ACTION Initialize:
// set interface array instances
aTestItems[ii] := ADR(fbTestFileLog);		ii := ii + 1;
aTestItems[ii] := ADR(fbTestSystemInfo); 	ii := ii + 1;
aTestItems[ii] := ADR(fbTestStation); 		ii := ii + 1;

//aTestItems[ii] := ADR(fbTestpid..);	ii := ii + 1;

bInitDone := TRUE;
END_ACTION

END_PROGRAM

// ---- Background/UnitTest/TestCases/Base/FB_TestCaseBase.TcPOU
/// Test case template
FUNCTION_BLOCK INTERNAL FB_TestCaseBase IMPLEMENTS ITestCase
VAR
	/// state of test case
	eState	: E_TestCaseState;
	/// result of test case
	eResult	: E_TestResult;
END_VAR

{attribute 'object_name' := 'Reset'}
METHOD Reset
// reset var's
eState := E_TestCaseState.eTestCaseState_ready;
eResult := E_TestResult.eTestResult_none;
END_METHOD

{attribute 'object_name' := 'Run'}
METHOD Run : E_TestCaseState
// set state to running, if ready
IF eState = E_TestCaseState.eTestCaseState_ready AND eResult = E_TestResult.eTestResult_none THEN
	eState := E_TestCaseState.eTestCaseState_running;
ELSIF eState <> E_TestCaseState.eTestCaseState_running THEN
	eState := E_TestCaseState.eTestCaseState_error;
END_IF

Run := eState;
END_METHOD

{attribute 'monitoring' := 'call'}
PROPERTY TestResult : E_TestResult
GET
TestResult := eResult;
END_GET
END_PROPERTY

{attribute 'monitoring' := 'call'}
PROPERTY TestState : E_TestCaseState
GET
TestState := eState;
END_GET
END_PROPERTY

END_FUNCTION_BLOCK

// ---- Background/UnitTest/TestCases/FB_TestCase01FileLog.TcPOU
FUNCTION_BLOCK FB_TestCase01FileLog EXTENDS FB_TestCaseBase
VAR
	/// dependencies
	ILog: I_Logger;
	
	bTestOk : BOOL := FALSE;
	bAddInfo, bAddWarn, bAddErr : BOOL;
END_VAR

{attribute 'object_name' := 'Run'}
METHOD Run : E_TestCaseState
// init state in base
Run := SUPER^.Run();
IF Run <> E_TestCaseState.eTestCaseState_running THEN
	RETURN;
END_IF

// test
ILog := Services.ILog;

IF bAddInfo THEN
	bAddInfo := FALSE;
	ILog.AddLog('Test none log message', sSource, E_LogLevel.eLogLevel_none);
	ILog.AddLog('Test info log message', sSource, E_LogLevel.eLogLevel_info);
	//P_HMI_Controller.UpdateNotificationPrio(E_Notification.eNotification_generalInf, TRUE, "UnitTest: eNotification_generalInf", E_Priority.ePriority_info);

	//SUPER^.M_SetErrorEx1(stTextListGlobal.stText_NG_Station005,  // Grp
	//				stTextListGlobal.stText_ST005_Name, "Antrieb (+E2-XXU1)", TO_WSTRING(fbDrive[E_St005_Object_Drive.eSt005_Drive_Antrieb].sErrText), 
	//				E_NotificationMode.eNotificationMode_Auto);

END_IF

IF bAddWarn THEN
	bAddWarn := FALSE;
	ILog.AddLog('Test warning log message', sSource, E_LogLevel.eLogLevel_warn);
	//P_HMI_Controller.UpdateNotificationPrio(E_Notification.eNotification_generalWarn, TRUE, "UnitTest: eNotification_generalWarn", E_Priority.ePriority_warning);
END_IF

IF bAddErr THEN
	bAddErr := FALSE;
	ILog.AddLog('Test error log message', sSource, E_LogLevel.eLogLevel_err);
	//P_HMI_Controller.UpdateNotificationPrio(E_Notification.eNotification_generalErr, TRUE, "UnitTest: eNotification_generalErr", E_Priority.ePriority_fault);
END_IF

// update result and state
IF bTestOk	THEN
	bTestOk := FALSE;
	eResult := E_TestResult.eTestResult_ok; //check log files!
	eState := E_TestCaseState.eTestCaseState_finished;
	Run := eState;
END_IF
END_METHOD

END_FUNCTION_BLOCK

// ---- Background/UnitTest/TestCases/FB_TestCase02SystemInfo.TcPOU
FUNCTION_BLOCK FB_TestCase02SystemInfo EXTENDS FB_TestCaseBase
VAR
	stTestPlcSystemInfo: ST_PlcSystemInfo;
	bTestOk : BOOL := TRUE;
END_VAR

{attribute 'object_name' := 'Run'}
METHOD Run : E_TestCaseState
// init state in base
Run := SUPER^.Run();
IF Run <> E_TestCaseState.eTestCaseState_running THEN
	RETURN;
END_IF

// test
stTestPlcSystemInfo := Statics.stPlcSystemInfo;

// update result and state
IF bTestOk THEN
	eResult := E_TestResult.eTestResult_ok; //check stTestPlcSystemInfo
	eState := E_TestCaseState.eTestCaseState_finished;
END_IF

Run := eState;
END_METHOD

END_FUNCTION_BLOCK

// ---- Background/UnitTest/TestCases/FB_TestCase03Station.TcPOU
FUNCTION_BLOCK FB_TestCase03Station EXTENDS FB_TestCaseBase
VAR
	fbTestStation	: FB_TestStation;
	stTestStationIO : ST_TestStation_IO;
	eStState		: E_ComponentState;
	iTest			: INT;
	bInit			: BOOL;
	bEnable			: BOOL := TRUE;
	bSafetyOk		: BOOL := TRUE;
	bTestOk 		: BOOL := FALSE;
END_VAR

{attribute 'object_name' := 'Run'}
METHOD Run : E_TestCaseState
// init state in base
Run := SUPER^.Run();
IF Run <> E_TestCaseState.eTestCaseState_running THEN
	RETURN;
END_IF

// test
fbTestStation.Enable := bEnable;
fbTestStation.SafetyOk := bSafetyOk;
fbTestStation();
CASE iTest OF
	0:	// init / idle / no Test
		IF NOT bInit THEN
			iTest := 1;
			RETURN;
		END_IF
		
	10:	// init Station
		bInit := TRUE;
		fbTestStation.stIO := stTestStationIO;		
		
	20:	// reset
		fbTestStation.Reset();
		
	30:	// execute command
		;//stRes := fbTestStation.ExecuteCmd(stCmd);
		
END_CASE
iTest := 0;

// update result and state
IF bTestOk THEN
	eResult := E_TestResult.eTestResult_ok; //check log files!
	eState := E_TestCaseState.eTestCaseState_finished;
END_IF

Run := eState;
END_METHOD

END_FUNCTION_BLOCK

// ---- Background/UnitTest/TestCases/StationTest/FB_TestStation.TcPOU
FUNCTION_BLOCK FB_TestStation EXTENDS FB_StationBase
VAR_INPUT
	// IO ref
	stIO	: REFERENCE TO ST_TestStation_IO;
END_VAR
VAR_OUTPUT
END_VAR
VAR
	// components
	fbAxis 		: FB_AxisDriver;
	fbCylinder 	: FB_Cylinder;
END_VAR

/// 
/// Station 01 function block 
/// TW/www.rmth.at/09.2016
///

ACTION DEMO:
(*
IF fbStepAuto.FirstShotSequence THEN
	; //Diese Aktion wird erstmals aufgerufen. Beispiel: zum Initilisieren der Aktion...
END_IF
*)
///		---------------------------------------------	PROCESS   ---------------------------------------------		
(*
CASE iStepAuto OF
	
	0:	aSClearText[EN] := 'PROCESS: wait for enable';
		aSClearText[DE] := 'PROCESS: warte auf Freigabe';
		IF bStepTrigger THEN
			; //Dieser Schritt wird erstmals aufgerufen. Beispiel: zum Initilisieren des akt. Schritts
		END_IF

		IF tonStep.ET > T#1S THEN // Beispiel Schrittverzögerung (1 Sekunde)
			iStepAuto := 10;
		END_IF
		
	10:	aSClearText[EN] := 'PROCESS: demo move';
		aSClearText[DE] := 'PROCESS: Demo move';
		CycleStart();
		IF RunStep THEN // RunStep immer vor Bewegungen (Zylinder, Servo, Robot,..) abfragen!!!
			// fbServo.MoveTo(1200);
			iStepAuto := 20;
		END_IF
	
	20:	aSClearText[EN] := 'PROCESS: demo condition, message';
		aSClearText[DE] := 'PROCESS: Demo Abfrage, Meldung';
		//IF fbServo.TargetReached THEN
			iStepAuto := 30;
		//ELSIF fbSequence.tonStep.ET > T#10S THEN
			SetError('Servo Zielposition wurde nicht erreicht.');	//SetInfo(... SetWarning(...
			//UpdateInfo(... UpdateWarning(... UpdateError(...  
		//END_IF
		
	30:	aSClearText[EN] := 'PROCESS: demo logging system';
		aSClearText[DE] := 'PROCESS: Demo Logging-System';
		//IF bDebugLog THEN			
			AddLogInf(Concat2x('Servo Amplifier Temp: ', '75')); //LREAL_TO_STRING(fbAxisDriver.AmplifierTemp)));	
			//AddLogWrn(..
			//AddLogErr(..
		//END_IF
		iStepAuto := 40;
		
	40:	aSClearText[EN] := 'PROCESS: demo statics/system info';
		aSClearText[DE] := 'PROCESS: Demo STATICS/SystemInfos';
		// aktuelle Zeit: dtTime := Statics.dtNow; // aktuelle Zeit als String: Statics.sTimeString
		// Farben: nstateColor := Statics.stColor.Green;
		// Impulse: Statics.stPulse.bImpulse500ms; Statics.stPulse.bImpulse300ms; ...
		// ToggleBits: bLed := Statics.stPulse.bToggle500ms;
		
		// Systeminformationen: Statics.stPlcSystemInfo.fCycleTime;
								//Statics.stPlcSystemInfo.fLastExecTime;
								//Statics.stPlcSystemInfo.stPlcAppSystemInfo.AdsPort;  Statics.stPlcSystemInfo.stPlcAppSystemInfo.OnlineChangeCnt; ...
								//Statics.stPlcSystemInfo.stPlcTaskSystemInfo.FirstCycle
		iStepAuto := 50;
		
	50: aSClearText[EN] := 'PROCESS: counter and timer!';
		aSClearText[DE] := 'PROCESS: Zaehler und Timer!';
		AddLogInf(Concat2x('Stationszyklen (Tag): ', UDINT_TO_STRING(diCycles)));
		AddLogInf(Concat2x('Stationszyklen (Ges): ', UDINT_TO_STRING(diTotalCycles)));
		AddLogInf(Concat2x('Zykluszeit Station [ms]: ', UDINT_TO_STRING(diLastCycleTime)));
		CycleEnd();
		iStepAuto := 10;

		
END_CASE
*)
END_ACTION

METHOD PROTECTED M_Homing
VAR
END_VAR
// Homing sequence
IF NOT bRunHoming THEN
	RETURN;
END_IF

// Homingablauf
CASE arriStepHome[0] OF
	
	0:	aSClearText := "HOMING: signal reset";
		arriStepHome[0] := 10;
		
	10:	aSClearText := "HOMING: wait for enable";
		IF RunStep THEN
			arriStepHome[0] := 20;
		END_IF
		
	20:	aSClearText := "HOMING: home position reached";
		IF arrtonStep[0].ET > T#1S THEN
			bRunHoming := FALSE;
			arriStepHome[0] := 0;	
		END_IF
		
END_CASE
END_METHOD

METHOD PROTECTED M_Manual
VAR_INPUT
END_VAR
// manual mode
IF NOT (eOpMode = eOpMode_manual) THEN
	RETURN;
END_IF

(*
CASE stManualCmd.iCommand OF
	// no command
	eStation01ManualCommand_none: RETURN;
	
	// cylinder HP/WP
	eStation01ManualCommand_cyl01Hp:
		aSClearText[EN] := 'last manual cmd: Cyl.01 HP';
		
	// cylinder HP/WP
	eStation01ManualCommand_cyl01Wp:
		aSClearText[EN] := 'last manual cmd: Cyl.01 WP';
	
		
END_CASE

/// delect command
MEMSET(ADR(stManualCmd), 0 , SIZEOF(stManualCmd)); *)
END_METHOD

METHOD PROTECTED M_Sequence
VAR
END_VAR
(*
IF fbStepAuto.FirstShotSequence THEN
	; //Diese Aktion wird erstmals aufgerufen. Beispiel: zum Initilisieren der Aktion...
END_IF
*)
///		---------------------------------------------	PROCESS   ---------------------------------------------		
CASE arriStepAuto[0] OF
	
	0:	aSClearText := "PROCESS: wait for enable";
		IF bStepTrigger THEN
			; //Dieser Schritt wird erstmals aufgerufen. Beispiel: zum Initilisieren des akt. Schritts
		END_IF

		IF arrtonStep0].ET > T#1S THEN // Beispiel Schrittverzögerung (1 Sekunde)
			arriStepAuto[0] := 10;
		END_IF
		
	10:	aSClearText := "PROCESS: demo move";
		CycleStart();
		IF RunStep THEN // RunStep immer vor Bewegungen (Zylinder, Servo, Robot,..) abfragen!!!
			// fbServo.MoveTo(1200);
			arriStepAuto[0] := 20;
		END_IF
	
	20:	aSClearText := "PROCESS: demo condition, message";
		//IF fbServo.TargetReached THEN
			arriStepAuto[0] := 30;
		//ELSIF fbSequence.tonStep.ET > T#10S THEN
			SetError("Servo Zielposition wurde nicht erreicht.");	//SetInfo(... SetWarning(...
			//UpdateInfo(... UpdateWarning(... UpdateError(...  
		//END_IF
		
	30:	aSClearText := "PROCESS: demo logging system";
		//IF bDebugLog THEN			
			AddLogInf(Concat2x('Servo Amplifier Temp: ', '75')); //LREAL_TO_STRING(fbAxisDriver.AmplifierTemp)));	
			//AddLogWrn(..
			//AddLogErr(..
		//END_IF
		arriStepAuto[0] :=  40;
		
	40:	aSClearText := "PROCESS: demo statics/system info";
		// aktuelle Zeit: dtTime := Statics.dtNow; // aktuelle Zeit als String: Statics.sTimeString
		// Farben: nstateColor := Statics.stColor.Green;
		// Impulse: Statics.stPulse.bImpulse500ms; Statics.stPulse.bImpulse300ms; ...
		// ToggleBits: bLed := Statics.stPulse.bToggle500ms;
		
		// Systeminformationen: Statics.stPlcSystemInfo.fCycleTime;
								//Statics.stPlcSystemInfo.fLastExecTime;
								//Statics.stPlcSystemInfo.stPlcAppSystemInfo.AdsPort;  Statics.stPlcSystemInfo.stPlcAppSystemInfo.OnlineChangeCnt; ...
								//Statics.stPlcSystemInfo.stPlcTaskSystemInfo.FirstCycle
		arriStepAuto[0] :=  50;
		
	50: aSClearText := "PROCESS: counter and timer!";
		AddLogInf(Concat2x('Stationszyklen (Tag): ', UDINT_TO_STRING(diCycles)));
		AddLogInf(Concat2x('Stationszyklen (Ges): ', UDINT_TO_STRING(diTotalCycles)));
		AddLogInf(Concat2x('Zykluszeit Station [ms]: ', UDINT_TO_STRING(diLastCycleTime)));
		CycleEnd();
		arriStepAuto[0] :=  10;

		
END_CASE
END_METHOD

END_FUNCTION_BLOCK

// ---- POUs/Plant/_Base/FB_StationBase.TcPOU
FUNCTION_BLOCK PUBLIC FB_StationBase EXTENDS FB_ComponentBase IMPLEMENTS IStation
VAR_INPUT
	/// Enable items
	bEmergencyStopOk 	: BOOL;
	bSafetyOk 			: BOOL;
	bEnable 			: BOOL;
	bAutoHome 			: BOOL;		// if its true station will be homed by start button
	iNumberOfStepChains	: INT := 1;	// count of stepchains per station
	iStepChainIndex		: INT; 		// index to link text of choosed stepchain to hmi
END_VAR
VAR_OUTPUT
	nStateColor			: DWORD;	// color for state of station
	bBusy				: BOOL;		// station is busy
	bTransferEnable		: BOOL;		// transfer enable from station
	stTextAuto			: ST_Text;	// T_MaxString;
	stTextHome			: ST_Text;	// T_MaxString;
	
	/// error-stop status
	bAutoStop_Error		: BOOL;
END_VAR
VAR
	/// Refs
	stHmiToStation		: REFERENCE TO ST_DefaultHmiToPlc;				// default hmi to station
	stHmiManualIn		: REFERENCE TO ST_HMI_BASE_STATION_MANUAL_IN;	// hmi manual to station
	stHmiManualOut		: REFERENCE TO ST_HMI_BASE_STATION_MANUAL_OUT;	// hmi manual from station
	stLocalSettings		: REFERENCE TO ST_StationDynSettings;			// dyn. station settings
	stLocalMonitoring	: REFERENCE TO ST_Monitoring_Station;			// dyn. station monitoring
	
	stLocalSettingsBackup	: ST_StationDynSettings;	// dyn. station settings
	
	/// private var's
	nStationNb		: INT;
	eStation		: E_Station;
	eParent 		: E_Module;
	eOpMode			: E_OpMode;	
	bStopped		: BOOL := TRUE;
	bTipEnable		: BOOL;
	
	/// enable var's
	bRunCycle, bRunStep, 
	bRunHoming, bInHome,
	bEnableManualStep		 : BOOL;

	/// counter
	diCycles				: UDINT; // Zykluszähler
	diLastCycleTime			: UDINT; // letzte Zykluszeit [ms]
	
	tonOpModeOff			: TON;
	fTrigSafetyOk			: F_TRIG;
	rtrigOpModeChanged		: R_TRIG;
		
	rtirgSafetyOpMode_Auto	: R_TRIG;
	rtirgSafetyOpMode_Hand	: R_TRIG;
	rtirgSafetyOpMode_Aus	: R_TRIG;
	
	bInitSettings	: BOOL;
	bInitMonitoring	: BOOL;
	bInitManual		: BOOL;
	
	sb				: FB_StringBuilder;
	sqHome, sqAuto	: FB_SequenceHelperSb;
	localEvents		: ST_DefaultEventClasses;
END_VAR
VAR PERSISTENT
	diTotalCycles	: UDINT; // Zykluszähler
	eOpModeOld		: E_OpMode;
END_VAR

/// 
/// Station 01 function block 
///

{attribute 'monitoring' := 'call'}
PROPERTY Busy : BOOL
GET
Busy := bBusy;
END_GET
END_PROPERTY

METHOD PROTECTED CycleEnd
VAR_INPUT
END_VAR
diCycles := diCycles + 1;
diTotalCycles := diTotalCycles + 1;
diLastCycleTime := TIME_TO_UDINT(sqAuto.SeqTime);
sqAuto.StopSequence();
bBusy := FALSE;
bStopped := TRUE;
END_METHOD

{attribute 'monitoring':='call'}
PROPERTY PUBLIC Cycles : UDINT
GET
Cycles := diCycles;
END_GET
SET
diCycles := Cycles;
END_SET
END_PROPERTY

METHOD PROTECTED CycleStart
VAR_INPUT
END_VAR
sqAuto.StartSequence();
bBusy := TRUE;
bStopped := FALSE;
END_METHOD

{attribute 'monitoring':='call'}
PROPERTY PUBLIC EmergencyStopOk : BOOL
GET
EmergencyStopOk := bEmergencyStopOk;
END_GET
SET
bEmergencyStopOk := EmergencyStopOk;
END_SET
END_PROPERTY

{attribute 'monitoring':='call'}
PROPERTY PUBLIC Enable : BOOL
GET
Enable := bEnable;
END_GET
SET
bEnable := Enable;
END_SET
END_PROPERTY

{attribute 'monitoring':='call'}
//{attribute 'monitoring' := 'variable'}
PROPERTY PUBLIC EnableManual : BOOL
GET
EnableManual := EnableSummary AND (eOpMode = eOpMode_manual);
END_GET
END_PROPERTY

{attribute 'monitoring':='call'}
//{attribute 'monitoring' := 'variable'}
PROPERTY INTERNAL EnableSummary : BOOL
GET // PUBLIC
EnableSummary := bEnable 
				AND bSafetyOk 
				AND (bRunHoming OR (eOpMode = eOpMode_manual) OR (eOpMode = eOpMode_step) OR (eOpMode = eOpMode_auto));
END_GET
END_PROPERTY

METHOD PROTECTED GetComponentError : I_StringBuilder
VAR_IN_OUT
	fbUi	: FB_ManualUiBase;
END_VAR
VAR
	tmp		: ST_Text;
	name,
	err, 
	bmk		: STRING;
END_VAR
WSTRING_TO_STRING2(ADR(name), ADR(fbUi.stName.wsName), SIZEOF(name));		//ToDo: get rid of wstring?
WSTRING_TO_STRING2(ADR(err), ADR(fbUi.stErrorText.wsName), SIZEOF(err));
WSTRING_TO_STRING2(ADR(bmk), ADR(fbUi.stBmk.wsName), SIZEOF(bmk));

GetComponentError := sb.Set(name)
  .Append(' | ')  
  .Append(err)
  .Append(' | ')
  .Append(bmk);
END_METHOD

METHOD PUBLIC GetStepChainTest : ST_Text
VAR_INPUT
	Index : INT; // step chain index
END_VAR
// step chain index is ignored in the default implementation -> if multiple step chains are needed, use derived base and override this method. 
GetStepChainTest.nNameId := sqAuto.InfoTextId;
GetStepChainTest.wsName := sqAuto.Info.ToWString();
GetStepChainTest.wsNameId := sqAuto.InfoTextWsId;
END_METHOD

{attribute 'monitoring':='call'}
PROPERTY PUBLIC Homing : BOOL
GET
Homing := bRunHoming;
END_GET
END_PROPERTY

/// Station in Home flag
{attribute 'monitoring':='call'}
PROPERTY InHome : BOOL
GET
InHome := TRUE;
//FOR ii := 0 TO iNumberOfStepChains - 1 DO
	IF NOT sqHome.InHome THEN
		InHome := FALSE;
	END_IF
//END_FOR

bInHome := InHome;
IF InHome THEN
	bRunHoming := FALSE;
END_IF
END_GET
END_PROPERTY

METHOD PUBLIC InitEvents : IStation
VAR_IN_OUT CONSTANT
	infoEvent,
	warnEvent,
	errorEvent : TcEventEntry;
END_VAR
// create default station alarms
localEvents.Info := infoEvent;
localEvents.Warning := warnEvent;
localEvents.Error := errorEvent;
IEvent.CreateAlarm(infoEvent, FALSE, TcSourceInfo)
	  .CreateAlarm(warnEvent, TRUE, TcSourceInfo)
	  .CreateAlarm(errorEvent, TRUE, TcSourceInfo);

InitEvents := THIS^;
END_METHOD

METHOD PROTECTED M_CallObjects : BOOL
VAR_INPUT
END_VAR
// Call objects - to be subclassed
END_METHOD

METHOD PROTECTED M_DynMonitoring : BOOL
VAR_INPUT
END_VAR
// station base signals
stLocalMonitoring.bInHome := bInHome;
stLocalMonitoring.bAuto := bRunStep;
stLocalMonitoring.bBusy := bBusy;
stLocalMonitoring.bError := (eState = E_ComponentState.eComponentState_error);
stLocalMonitoring.bManual := (eOpMode = E_OpMode.eOpMode_manual);
stLocalMonitoring.bTransferEnable := bTransferEnable;
stLocalMonitoring.bWarning := (eState = E_ComponentState.eComponentState_warning);

M_DynMonitoring := TRUE;
END_METHOD

METHOD PUBLIC M_EnableSummary : BOOL
VAR_INPUT
END_VAR
END_METHOD

METHOD PROTECTED M_Homing
VAR
END_VAR
// Homing sequence - to be subclassed
END_METHOD

METHOD PUBLIC M_Init : IStation
VAR_INPUT
END_VAR
// set up defaults
Active := TRUE;
Enable := TRUE;
SUPER^.M_InitComponentBase();

// set up station id and name -> to be subclassed... 
//Station := E_Station.eStation_none;
//stName := stTextListGlobal.stText_ST000_Name;

sqAuto.SetInfo(Name);
nStateColor := TO_DWORD(STATICS.stColor.White);

stHmiToStation REF= P_HMI_Controller.aStHmiToStation[eStation];
stHmiManualIn REF= HMI.stHmi.stIn.arrStStation[eStation].stManual;
stHmiManualOut REF= HMI.stHmi.stOut.stCommon.arrStStation[eStation].stManual;
stLocalSettings REF= Services.stSettings.stStationSettings[eStation];
stLocalMonitoring REF= HMI.stHmi.stOut.stCommon.stMonitoring.astMonitoringStation[eStation];

//FOR ii := 0 TO CONST.iMaxIdxLocalStepChain DO
	sqAuto.SetInfo(stTextListGlobal.stText_initialize_station);	// -> to be subclassed, ... 
//END_FOR

M_Init := THIS^;
END_METHOD

METHOD PROTECTED M_InitDynManual : BOOL
VAR_INPUT
	nIndex			: INT;
	stName			: ST_Text;
	stGroup			: ST_Text;
	stType			: ST_Text;
	diObjectIndex	: DINT;
END_VAR
// chk
IF nIndex < 0 OR nIndex > CONST.iMaxIdxObject THEN
	StationError.ArgSbAppendRaise('Dyn. manual index out of range.');
	RETURN;
END_IF

stHmiManualOut.stObjects[nIndex].stName := stName;
stHmiManualOut.stObjects[nIndex].stGroup := stGroup;
stHmiManualOut.stObjects[nIndex].stType := stType;
stHmiManualOut.stObjects[nIndex].diObjectIndex := diObjectIndex;

M_InitDynManual := TRUE;
END_METHOD

METHOD PROTECTED M_InitDynManualUi : BOOL
VAR_IN_OUT
	fbManualUi	: FB_ManualUiBase;
END_VAR
VAR
	IManualUi	: I_ManualUi;
	nIx, ix		: INT;
END_VAR
IManualUi := fbManualUi;

// search next free index
nIx := -1;
FOR ix := 0 TO CONST.iMaxIdxObject DO
	IF stHmiManualOut.stObjects[ix].stName.wsName = "" THEN
		nIx := ix;
		EXIT;
	END_IF
END_FOR

IF nIx < 0 THEN
	StationError.ArgSbAppendRaise('Next free dyn. manual index not found.');
	RETURN;
END_IF

IManualUi.ObjectIndex := (StationNb * 1000) + nIx + 1; // create unique object index

M_InitDynManualUi := M_InitDynManual(nIx,			// index 
		IManualUi.Name,								// device name
		Name,										// group -> station name
		stTextListGlobal.stText_ObjectTypeDrive,	// type
		IManualUi.ObjectIndex);						// object index
		
IManualUi.M_SetStateObject(stHmiManualOut.stObjects[nIx]);
END_METHOD

METHOD PROTECTED M_InitDynMonitoringItem : BOOL
VAR_INPUT
	nIndex		: INT;
	wsName		: WSTRING;
	stGroup		: ST_Text;
	eDataType	: E_DataType;
	stUnit		: ST_Text;			
END_VAR
// chk
IF nIndex < 0 OR nIndex > CONST.iMaxIdxMonitoring THEN
	StationError.ArgSbAppendRaise('Dyn. monitoring index out of range.');
	RETURN;
END_IF

stLocalMonitoring.astMonitoring[nIndex].stIndex.nNameId := nIndex;
stLocalMonitoring.astMonitoring[nIndex].stIndex.wsNameId := wsName;
stLocalMonitoring.astMonitoring[nIndex].stName := F_CreateDynText(wsName, nIndex);
stLocalMonitoring.astMonitoring[nIndex].eDataType := eDataType;
stLocalMonitoring.astMonitoring[nIndex].stGroup := stGroup;
stLocalMonitoring.astMonitoring[nIndex].stUnit := stUnit;

M_InitDynMonitoringItem := TRUE;
END_METHOD

METHOD PROTECTED M_InitDynSettingsItem : BOOL
VAR_INPUT
	nIndex					: INT;
	wsIndex					: WSTRING;
	stSettGroup				: ST_Text;
	stSettTitle				: ST_Text;
	stSettUnit				: ST_Text;	
	eSettDataType			: E_DataType;	
	fSettValueMin			: REAL;
	fSettValueMax			: REAL;
	// required user level, 0 = none
	nRequiredUserLevel		: INT := 0;	
END_VAR
// chk
IF nIndex < 0 OR nIndex > CONST.iMaxIdxLocalSetting THEN
	StationError.ArgSbAppendRaise('Dyn. setting index out of range.');
	RETURN;
END_IF

M_InitDynSettingsItem := F_InitDynDataItem(
							nIndex,
							wsIndex,
							stSettGroup,
							stSettTitle,
							stSettUnit,
							eSettDataType,
							fSettValueMin,
							fSettValueMax,
							// required user level, 0 = none
							nRequiredUserLevel,
							E_RecipeMode.eRecipeMode_ToFrom,
							stLocalSettings.stDynStationSettings);
END_METHOD

METHOD PUBLIC M_InitEx : IStation
VAR_INPUT
	ILogger			: I_Logger;
	IEventHandler	: I_EventHandler;
END_VAR
M_InitEx := THIS^.M_Init();

// set up logger and event handler
SUPER^.M_InitComponentBaseEx(ILogger, IEventHandler);

// init extended stuff here...
END_METHOD

METHOD M_InitSequences : BOOL
VAR_INPUT
END_VAR
sqHome.Reset();
sqAuto.Reset(); 
sqAuto.SetInfo(stTextListGlobal.stText_initialize_station);
END_METHOD

METHOD PROTECTED M_Manual
VAR_INPUT
END_VAR
// Manual mode - to be subclassed
END_METHOD

METHOD PROTECTED M_OpModeChanged : BOOL
VAR_INPUT
END_VAR
// to be subclassed
END_METHOD

METHOD PUBLIC M_Run : BOOL
VAR
END_VAR
M_Run := TRUE; // to be subclassed..

// call component run
SUPER^.Run();

// Safety OP-Mode
rtirgSafetyOpMode_Auto(CLK := stHmiToStation.eSafetyOpMode = E_Opmode.eOpMode_auto);
rtirgSafetyOpMode_Hand(CLK := stHmiToStation.eSafetyOpMode = E_Opmode.eOpMode_manual);
rtirgSafetyOpMode_Aus(CLK := stHmiToStation.eSafetyOpMode = E_Opmode.eOpMode_off);

// reset (all or this station)
IF stHmiToStation.bReset THEN
	Reset();
END_IF

// step (all or this station)
// step -> ist bei Auto über die Property immer TRUE
bRunStep := stHmiToStation.bStep;
	
// start (all or this station)
IF stHmiToStation.bStart OR P_Safety.bMachineRequestStart OR stHmiToStation.bStep THEN		
	IF NOT bEnable THEN
		StationWarning.ArgSetString('Kein Enable Signal bei Start').Raise();
	ELSIF NOT bSafetyOk THEN
		StationWarning.ArgSetString('Safety nicht ok bei Start').Raise();
	// Fehler steht noch an
	ELSIF bAutoStop_Error THEN
		StationWarning.ArgSetString('Station in Fehlerstatus --> Reset').Raise();

	// Safety muss in Auto sein
	ELSIF stHmiToStation.eSafetyOpMode <> E_Opmode.eOpMode_auto AND Const.bEnSafetyOpMode THEN
		StationWarning.ArgSetString('Safety Betriebsart nicht AUTO').Raise();
		
	// START
	ELSIF (OpMode = E_Opmode.eOpMode_auto OR OpMode = E_Opmode.eOpMode_step) THEN
		//bRunStep := FALSE;
		bRunCycle := TRUE;
	END_IF
END_IF

// cycle stop (all or this station)
IF stHmiToStation.bStop OR P_Safety.bMachineRequestCycleStop OR P_Supervision.bCycleStop THEN
	bRunCycle := bRunHoming := FALSE;
END_IF

// fast stop (all or this station)
IF stHmiToStation.bFastStop OR P_Supervision.bFastStop THEN 
	bRunCycle := bRunStep := bRunHoming := FALSE;
END_IF

// set op mode (all or this station)
tonOpModeOff(IN := stHmiToStation.bStop, PT := T#10S);
IF stHmiToStation.bOpModeManual OR rtirgSafetyOpMode_Hand.Q THEN
	bRunStep := FALSE;
	bRunCycle := FALSE;
	bRunHoming := FALSE;
	eOpMode := E_OpMode.eOpMode_manual;
ELSIF stHmiToStation.bOpModeAuto OR rtirgSafetyOpMode_Auto.Q THEN
	bRunStep := FALSE;
	bRunCycle := FALSE;
	bRunHoming := FALSE;
	eOpMode := E_OpMode.eOpMode_auto;
ELSIF stHmiToStation.bOpModeStep THEN
	bRunStep := FALSE;
	bRunCycle := FALSE;
	bRunHoming := FALSE;
	eOpMode := E_OpMode.eOpMode_step;
ELSIF tonOpModeOff.Q THEN
	eOpMode := E_OpMode.eOpMode_off;
END_IF
	
IF NOT bEmergencyStopOk THEN
	sqHome.InHome := FALSE;
	sqHome.Step := 0;
	sqAuto.Step := 0;
END_IF

// homing (all or this station)
IF stHmiToStation.bHome OR (stHmiToStation.bStart AND bAutoHome AND NOT sqHome.InHome AND sqHome.Step = 0 AND sqAuto.Step = 0) THEN
	IF NOT bEnable THEN
		StationWarning.ArgSbAppendRaise('Kein Enable Signal bei Start Grundstellung');
	ELSIF NOT bSafetyOk THEN
		StationWarning.ArgSbAppendRaise('Safety nicht ok bei Start Grundstellung');
		
	// Fehler steht noch an
	ELSIF bAutoStop_Error THEN
		StationWarning.ArgSbAppendRaise('Station in Fehlerstatus --> Reset');
	ELSE		
		sqHome.Step := 0;
		sqHome.InHome		:= FALSE;
		bRunCycle			:= FALSE;
		bRunHoming 			:= TRUE;
	END_IF
END_IF

/// Set Station State Color
IF State = eComponentState_error THEN
	nStateColor := STATICS.stColor.Red;
ELSIF bInHome AND (eOpMode = eOpMode_Auto OR eOpMode = eOpMode_Step) THEN	
	nStateColor := STATICS.stColor.LightBlue;
ELSIF bStopped AND (eOpMode = eOpMode_Auto OR eOpMode = eOpMode_Step) THEN
	nStateColor := STATICS.stColor.Blue;									
ELSIF State = eComponentState_running AND (eOpMode = eOpMode_Auto OR eOpMode = eOpMode_Step) THEN
	nStateColor := STATICS.stColor.LimeGreen;					
ELSIF State = eComponentState_running AND eOpMode = eOpMode_manual THEN
	nStateColor := STATICS.stColor.Orange;		
ELSE
	nStateColor := STATICS.stColor.White;
END_IF

//StepChainTextMapping
//stTextAuto := arraSTextAuto[iStepChainIndex];
//IF iStepChainIndex >= 0 AND iStepChainIndex <= CONST.iMaxIdxLocalStepChain THEN
	stTextAuto.nNameId := sqAuto.InfoTextId;
	stTextAuto.wsName := WConcat3(TO_WSTRING(sqAuto.Step),": ", sqAuto.Info.ToWString());
	stTextAuto.wsNameId := WConcat3(TO_WSTRING(sqAuto.Step),": ", sqAuto.InfoTextWsId);	
	
	//stTextHome := arraSTextHome[iStepChainIndex];
	stTextHome.nNameId := sqHome.InfoTextId;
	stTextHome.wsName := WConcat3(TO_WSTRING(sqHome.Step), ": ", sqHome.Info.ToWString());
	stTextHome.wsNameId := WConcat3(TO_WSTRING(sqHome.Step),": ", sqHome.InfoTextWsId);
//END_IF

rtrigOpModeChanged(CLK := eOpModeOld <> eOpMode);
IF rtrigOpModeChanged.Q THEN
	eOpModeOld := eOpMode;
	M_OpModeChanged();
END_IF

//call methodes
sqHome.EnableStep := RunStep;
sqHome();
sqAuto.EnableStep := RunStep;
sqAuto();

M_CallObjects();
M_Homing();
M_Sequence();
M_Manual();
M_Supervision();
END_METHOD

METHOD PROTECTED M_Sequence
VAR
END_VAR
// Automatic sequence - to be subclassed
END_METHOD

METHOD PROTECTED M_Supervision : BOOL
VAR_INPUT
END_VAR
// to be subclassed
END_METHOD

/// Station OP Mode
{attribute 'monitoring':='call'}
PROPERTY OpMode : E_OpMode
GET
OpMode := eOpMode;
END_GET
END_PROPERTY

{attribute 'monitoring':='call'}
PROPERTY Parent : E_Module
GET
Parent := eParent;
END_GET
END_PROPERTY

METHOD PROTECTED ReactToComponentError
VAR_IN_OUT
	fbUi	: FB_ManualUiBase;
END_VAR
VAR_INPUT
	mode 	: E_EventReaction;
END_VAR
VAR
	msg		: I_StringBuilder;
END_VAR
msg := GetComponentError(fbUi);
ReactToEvent(mode, TcEventSeverity.Error)
			.ArgSetSbRaise(msg);
END_METHOD

METHOD PROTECTED ReactToError : I_EventHandler
VAR_INPUT
	mode : E_EventReaction;
END_VAR
ReactToError := ReactToEvent(mode, TcEventSeverity.Error);
END_METHOD

METHOD PROTECTED ReactToEvent : I_EventHandler
VAR_INPUT
	mode		: E_EventReaction;
	severity	: TcEventSeverity;
END_VAR
// switch event reaction mode
CASE mode OF
	E_EventReaction.Init:
		M_InitSequences();
		
	E_EventReaction.Stop:
		bRunCycle := FALSE;
		bAutoStop_Error := TRUE;
		
	E_EventReaction.CycleStop:
		bRunCycle := FALSE;
		
END_CASE

// set the component state &
//  return value (info, warning or error - event handler)
CASE severity OF
	TcEventSeverity.Info:
		eState := E_ComponentState.eComponentState_info;
		ReactToEvent := StationInfo;
		
	TcEventSeverity.Warning:
		eState := E_ComponentState.eComponentState_warning;
		ReactToEvent := StationWarning;
		
	ELSE
		eState := E_ComponentState.eComponentState_error;
		ReactToEvent := StationError;
		
END_CASE
END_METHOD

METHOD PROTECTED ReactToInfo : I_EventHandler
VAR_INPUT
	mode : E_EventReaction;
END_VAR
ReactToInfo := ReactToEvent(mode, TcEventSeverity.Info);
END_METHOD

METHOD PROTECTED ReactToWarn : I_EventHandler
VAR_INPUT
	mode : E_EventReaction;
END_VAR
ReactToWarn := ReactToEvent(mode, TcEventSeverity.Warning);
END_METHOD

/// Reset component logic
{attribute 'object_name' := 'Reset'}
METHOD Reset
VAR
	iIdxSub			: INT;
END_VAR
// base logic run
SUPER^.Reset();

// reset var's
nStateColor := STATICS.stColor.White;

bAutoStop_Error := FALSE;
END_METHOD

{attribute 'monitoring':='call'}
PROPERTY PUBLIC RunCycle : BOOL
GET // PUBLIC
RunCycle := bRunCycle;
END_GET
SET // PUBLIC
bRunCycle := RunCycle;
END_SET
END_PROPERTY

{attribute 'monitoring':='variable'}
PROPERTY PUBLIC RunManStep : Bool
GET
RunManStep := EnableSummary AND
			NOT bAutoStop_Error AND
			(OpMode = E_OpMode.eOpMode_manual AND (bRunStep OR NOT bEnableManualStep));
END_GET
END_PROPERTY

{attribute 'monitoring':='variable'}
PROPERTY PUBLIC RunStep : BOOL
GET
VAR
	sMsg : WSTRING(255);
END_VAR
// Rückgabe
RunStep := EnableSummary AND
			NOT bAutoStop_Error AND
			((bRunStep AND eOpMode = eOpMode_step) OR
			(eOpMode = eOpMode_auto));
END_GET
END_PROPERTY

{attribute 'monitoring':='call'}
PROPERTY PUBLIC SafetyOk : BOOL
GET
SafetyOk := bSafetyOk;
END_GET
SET
bSafetyOk := SafetyOk;
END_SET
END_PROPERTY

{attribute 'monitoring':='call'}
PROPERTY StateColor : DWORD
GET
StateColor := nStateColor;
END_GET
END_PROPERTY

{attribute 'monitoring':='call'}
PROPERTY PUBLIC Station : E_Station
GET
Station := eStation;
END_GET
SET // PUBLIC
eStation := Station;
END_SET
END_PROPERTY

PROPERTY PROTECTED StationError : I_EventHandler
GET
// return the event handler
//	prepare string builder w. station info
StationError := IEvent.Select(localEvents.Error)
					  .ArgSbInitWs(stName.wsName)
					  .ArgSbAppend(' | ');
END_GET
END_PROPERTY

PROPERTY PROTECTED StationInfo : I_EventHandler
GET
// return the event handler
//	prepare string builder w. station info
StationInfo := IEvent.Select(localEvents.Info)
					 .ArgSbInitWs(stName.wsName)
					 .ArgSbAppend(' | ');
END_GET
END_PROPERTY

PROPERTY PUBLIC StationNb : INT
GET
StationNb := nStationNb;
END_GET
SET // PUBLIC
nStationNb := StationNb;
END_SET
END_PROPERTY

PROPERTY PROTECTED StationWarning : I_EventHandler
GET
// return the event handler
//	prepare string builder w. station info
StationWarning := IEvent.Select(localEvents.Warning)
					 .ArgSbInitWs(stName.wsName)
					 .ArgSbAppend(' | ');
END_GET
END_PROPERTY

/// Station stopped
{attribute 'monitoring':='call'}
PROPERTY Stopped : BOOL
GET
Stopped := bStopped;
END_GET
END_PROPERTY

PROPERTY TextAuto : ST_Text
GET
TextAuto := stTextAuto;
END_GET
END_PROPERTY

PROPERTY TextHome : ST_Text
GET
TextHome := stTextHome;
END_GET
END_PROPERTY

{attribute 'monitoring':='call'}
PROPERTY PUBLIC TipEnable : BOOL
GET
TipEnable := bTipEnable;
END_GET
END_PROPERTY

{attribute 'monitoring':='call'}
PROPERTY PUBLIC TotalCycles : UDINT
GET
TotalCycles := diTotalCycles;
END_GET
END_PROPERTY

{attribute 'monitoring' := 'call'}
PROPERTY TransferEnable : BOOL
GET
TransferEnable := bTransferEnable;
END_GET
END_PROPERTY

END_FUNCTION_BLOCK

// ---- POUs/Components/_Base/FB_ComponentBase.TcPOU
/// Abstract base FB for components
{attribute 'enable_dynamic_creation' := ''}
{attribute 'reflection' := ''}
FUNCTION_BLOCK FB_ComponentBase IMPLEMENTS ITFComponent
VAR
	ii				: INT;
	/// Unique ID of this instance (cam be used as index: P_ComponentPool.aComponents[iID]...)
	iId				: INT;
	/// component type
	eTyp			: E_ComponentType;
	/// component active flag
	bActive			: BOOL;
	/// component state
	eState			: E_ComponentState;
	// Logger
	ILog			: I_Logger;
	/// path of this FB (e.g. for log: P_ComponentPool.fbVirtualMaster)	
    {attribute 'instance-path'} 
    {attribute 'noinit'}
    {attribute 'hide'} 
	sPath			: STRING;
	// object id
	wsObjectId		: WSTRING;

	/// component name
	stName			: ST_Text;
	/// component name
	sBMK			: STRING;
	/// clear text info
	//aSClearText		: ARRAY[0..eLanguage_maxIdx] OF T_MaxString;
	aSClearText		: ST_Text;//T_MaxString;
	
	/// last error debug info
	sLastError		: T_MaxString;
	
	// event handler & source info
	IEvent			: I_EventHandler;
	TcSourceInfo	: FB_TcSourceInfo;
END_VAR

///
/// Abstract base FB for components
/// TP/www.rmth.at/11.2014
///

/// Get's or set's a value indicating whether this component is active or not.
{attribute 'monitoring':='call'}
PROPERTY Active : BOOL
GET
Active := bActive;
END_GET
SET
bActive := Active;
aSClearText := F_CreateDynTextDefaultS(SEL(bActive, 'INACTIVE!', 'ACTIVE!'));
END_SET
END_PROPERTY

METHOD PROTECTED AddLogErr
VAR_INPUT
	sLog : T_MaxString;
END_VAR
// chk
IF ILog = 0 THEN
	RETURN;
END_IF

ILog.AddLog(sLog, WSTRING_TO_STRING(stName.wsName), E_LogLevel.eLogLevel_err);
END_METHOD

METHOD PROTECTED AddLogInf
VAR_INPUT
	sLog : T_MaxString;
END_VAR
// chk
IF ILog = 0 THEN
	RETURN;
END_IF

ILog.AddLog(sLog, WSTRING_TO_STRING(stName.wsName), E_LogLevel.eLogLevel_info);
END_METHOD

METHOD PROTECTED AddLogWrn
VAR_INPUT
	sLog : T_MaxString;
END_VAR
VAR

END_VAR
// chk
IF ILog = 0 THEN
	RETURN;
END_IF

ILog.AddLog(sLog, WSTRING_TO_STRING(stName.wsName), E_LogLevel.eLogLevel_warn);
END_METHOD

{attribute 'monitoring':='call'}
PROPERTY BMK : STRING
GET
BMK := sBMK;
END_GET
SET
sBMK := BMK;
END_SET
END_PROPERTY

/// Get's value representing the component state.
{attribute 'monitoring':='call'}
PROPERTY ClearText : WSTRING(255)
GET
ClearText := aSClearText.wsName;
END_GET
END_PROPERTY

/// Unique component ID (cam be used as index: P_ComponentPool.aComponents[eID]...)
{attribute 'monitoring':='call'}
PROPERTY ID : INT
GET
ID := iId;
END_GET
SET
iId := ID;
END_SET
END_PROPERTY

/// Get's value representing the component state.
{attribute 'monitoring':='call'}
PROPERTY LastError : T_MaxString
GET
LastError := sLastError;
END_GET
END_PROPERTY

PROPERTY Logger : I_Logger
SET
ILog := Logger;
END_SET
END_PROPERTY

METHOD M_InitComponentBase : BOOL
VAR_INPUT
END_VAR
// set up default logger and event handler
ILog := Services.ILog;
IEvent := Services.fbEventHandler;
END_METHOD

METHOD M_InitComponentBaseEx : BOOL
VAR_INPUT
	ILogger			: I_Logger;
	IEventHandler	: I_EventHandler;
END_VAR
ILog := ILogger;
IEvent := IEventHandler;
END_METHOD

PROPERTY Name : ST_Text
GET
Name := stName;
END_GET
SET
stName := Name;
END_SET
END_PROPERTY

PROPERTY PUBLIC NameString : WSTRING(255)
GET
NameString := stName.wsName;
END_GET
END_PROPERTY

PROPERTY ObjectId : WSTRING
GET
ObjectId := wsObjectId;
END_GET
END_PROPERTY

{attribute 'monitoring':='call'}
PROPERTY Path : String
GET
Path := sPath;
END_GET
END_PROPERTY

PROPERTY RefsValid : BOOL
GET
RefsValid := IEvent <> 0;
END_GET
END_PROPERTY

/// Reset component logic
{attribute 'object_name' := 'Reset'}
METHOD Reset
/// abstract base logic reset

sLastError := sEmpty;

// default: set state to ready
eState := E_ComponentState.eComponentState_ready;
END_METHOD

/// Run component logic
{attribute 'object_name' := 'Run'}
METHOD Run : E_ComponentState
VAR
	ii : INT;
END_VAR
/// abstract base logic run

wsObjectId := TO_WSTRING( F_CutInstancePath(sPath) );

// only rdy state may lead to run
IF eState = E_ComponentState.eComponentState_ready THEN
	eState := E_ComponentState.eComponentState_running;
END_IF

Run := eState;
END_METHOD

/// Get's value representing the component state.
{attribute 'monitoring':='call'}
PROPERTY State : E_ComponentState
GET
State := eState;
END_GET
END_PROPERTY

/// Get's value representing the component state.
{attribute 'monitoring':='call'}
PROPERTY StateToString : STRING
GET
CASE eState OF

	eComponentState_none :
		StateToString := 'undefiniert';
	/// Component is resetting
	eComponentState_resetting:
		StateToString := 'wird zurückgesetzt';
	/// Component is ready
	eComponentState_ready:
		StateToString := 'ist bereit';
	/// Component is running
	eComponentState_running:
		StateToString := 'wird ausgeführt';
	/// Component has error
	eComponentState_error:
		StateToString := 'ist fehlerhaft';

END_CASE
END_GET
END_PROPERTY

{attribute 'monitoring':='call'}
PROPERTY Typ : E_ComponentType
GET
Typ := eTyp;
END_GET
END_PROPERTY

END_FUNCTION_BLOCK

// ---- POUs/HMI/Utilities/DynTxt/F_CreateDynTextDefaultS.TcPOU
FUNCTION F_CreateDynTextDefaultS : ST_Text
VAR_INPUT
	sText	: STRING;
END_VAR
VAR
END_VAR

F_CreateDynTextDefaultS.wsNameId := TO_WSTRING(sText);
F_CreateDynTextDefaultS.wsName := F_CreateDynTextDefaultS.wsNameId;

END_FUNCTION

// ---- POUs/System/Utilities/Functions/F_CutInstancePath.TcPOU
FUNCTION F_CutInstancePath : STRING(512)
VAR_INPUT
	sSrc			:STRING(512);
END_VAR
VAR
	sDelimiter		:STRING(1) := '.';
	iFnd			:UDINT;
	sSubstr			:STRING(512);
END_VAR

// sSrc := 'TE_SP_Module_Demo.TE_SP_Module_Demo_PlcRt1.P_MachineSet.fbMa2.fbDemoSequence.fbLenzei550';

iFnd := FIND2(ADR(sSrc), ADR(sDelimiter));
IF (iFnd > 0) THEN
	DELETE2(ADR(sSrc), ADR(sSubstr), SIZEOF(sSubstr), iFnd, 1);
END_IF
iFnd := FIND2(ADR(sSubstr), ADR(sDelimiter));
IF (iFnd > 0) THEN
	DELETE2(ADR(sSubstr), ADR(sSubstr), SIZEOF(sSubstr), iFnd, 1);
END_IF

F_CutInstancePath := sSubstr;

END_FUNCTION

// ---- POUs/System/Utilities/Sequencer/FB_SequenceHelperSb.TcPOU
FUNCTION_BLOCK FB_SequenceHelperSb EXTENDS FB_SequenceHelper
VAR_INPUT
END_VAR
VAR_OUTPUT
END_VAR
VAR
	wsb 			: FB_WStringBuilder;
	iInfoTextId		: INT;
	wsInfoTextId 	: WSTRING;
END_VAR

SUPER^();

PROPERTY PUBLIC Info : REFERENCE TO FB_WStringBuilder
GET
Info Ref= wsb;
END_GET
END_PROPERTY

PROPERTY PUBLIC InfoTextId : INT
GET
InfoTextId := iInfoTextId;
END_GET
SET
iInfoTextId := InfoTextId;
END_SET
END_PROPERTY

PROPERTY PUBLIC InfoTextWsId : WSTRING
GET
InfoTextWsId := wsInfoTextId;
END_GET
SET
wsInfoTextId := InfoTextWsId;
END_SET
END_PROPERTY

METHOD PUBLIC SetInfo : BOOL
VAR_INPUT
	stInfo : ST_Text;
END_VAR
iInfoTextId := stInfo.nNameId;
wsb.Set(stInfo.wsName);
wsInfoTextId := stInfo.wsNameId;
END_METHOD

END_FUNCTION_BLOCK

// ---- POUs/System/Utilities/Sequencer/FB_SequenceHelper.TcPOU
FUNCTION_BLOCK FB_SequenceHelper
VAR_INPUT
	InHome		: BOOL; // in home helper status flag
	Busy		: BOOL; // busy helper status flag
	EnableStep	: BOOL; // enable step mode
END_VAR
VAR_OUTPUT
	Init,				// step init flag
	SeqRun		: BOOL; // sequence run flag 
	StepTime,			// step time
	SeqTime		: TIME;	// sequence time
END_VAR
VAR
	nStep,
	nStepMirror	: UINT;
	tonStep,
	tonSequence	: TON;
END_VAR

Init := nStepMirror <> Step;
tonStep(IN := nStepMirror = Step, PT := T#49D17H2M47S295MS);
StepTime := tonStep.ET;
tonSequence(IN := SeqRun, PT := T#49D17H2M47S295MS);
SeqTime := tonSequence.ET;
nStepMirror := Step;

METHOD PUBLIC Reset : REFERENCE TO FB_SequenceHelper
VAR_INPUT
	value : UINT := 0;
END_VAR
Reset REF= THIS^;
Step := value;
END_METHOD

METHOD PUBLIC SetStep : REFERENCE TO FB_SequenceHelper
VAR_INPUT
	value : UINT;
END_VAR
SetStep REF= THIS^;

IF EnableStep THEN
	Step := value;	
END_IF
END_METHOD

METHOD PUBLIC StartSequence : REFERENCE TO FB_SequenceHelper
VAR_INPUT
END_VAR
StartSequence REF= THIS^;
tonSequence(IN := FALSE);
SeqRun := TRUE;
END_METHOD

{attribute 'monitoring' := 'call'}
PROPERTY PUBLIC Step : UINT
GET
Step := nStep;
END_GET
SET
nStep := Step;
END_SET
END_PROPERTY

METHOD PUBLIC StopSequence : REFERENCE TO FB_SequenceHelper
VAR_INPUT
END_VAR
StopSequence REF= THIS^;
SeqRun := FALSE;
END_METHOD

END_FUNCTION_BLOCK

// ---- POUs/System/Utilities/String/FB_WStringBuilder.TcPOU
FUNCTION_BLOCK FB_WStringBuilder IMPLEMENTS I_WStringBuilder
VAR_INPUT
END_VAR
VAR_OUTPUT
END_VAR
VAR
    wsString : WSTRING;
END_VAR

///
/// String Builder for WSTRING Fluent-Code Style
/// Credits to Gerhard Barteling, https://www.plccoder.com/fluent-code/
///

METHOD PUBLIC Append : I_WStringBuilder // Append text to the current build string.
VAR_INPUT
	text : WSTRING; // Text to append to current build string
END_VAR
wsString := WCONCAT(wsString, text);
Append := THIS^;
END_METHOD

METHOD PUBLIC AppendAny : I_WStringBuilder // Append text to the current build string.
VAR_INPUT
	value : ANY; // Value to append to current build string
END_VAR
VAR
	pSTR	: POINTER TO STRING;
	pWSTR	: POINTER TO WSTRING;
	pBOOL	: POINTER TO BOOL;
	pBYTE	: POINTER TO BYTE;
	pWORD	: POINTER TO WORD;
	pDWORD	: POINTER TO DWORD;
	pLWORD	: POINTER TO LWORD;
	pSINT	: POINTER TO SINT;
	pINT	: POINTER TO INT;
	pDINT	: POINTER TO DINT;
	pLINT	: POINTER TO LINT;
	pUSINT	: POINTER TO USINT;
	pUINT	: POINTER TO UINT;
	pUDINT	: POINTER TO UDINT;
	pULINT	: POINTER TO ULINT;
	pREAL	: POINTER TO REAL;
	pLREAL	: POINTER TO LREAL;
	pTIME	: POINTER TO TIME;
	pLTIME	: POINTER TO LTIME;
	pDATE	: POINTER TO DATE;
	pDT		: POINTER TO DT;
	pTOD	: POINTER TO TOD;
	pENUM	: POINTER TO ENUM;
END_VAR
CASE Value.TypeClass OF
	__SYSTEM.TYPE_CLASS.TYPE_STRING: 
		pSTR := value.pValue;
		wsString := WCONCAT(wsString, TO_WSTRING(pSTR^));
		
	__SYSTEM.TYPE_CLASS.TYPE_WSTRING:
		pWSTR := value.pValue;
		wsString := WCONCAT(wsString, TO_WSTRING(pWSTR^));
		
	__SYSTEM.TYPE_CLASS.TYPE_BOOL:
		pBOOL := value.pValue;
		wsString := WCONCAT(wsString, TO_WSTRING(pBOOL^));
		
	__SYSTEM.TYPE_CLASS.TYPE_BYTE:
		pBYTE := value.pValue;
		wsString := WCONCAT(wsString, TO_WSTRING(pBYTE^));
		
	__SYSTEM.TYPE_CLASS.TYPE_WORD:
		pWORD := value.pValue;
		wsString := WCONCAT(wsString, TO_WSTRING(pWORD^));
		
	__SYSTEM.TYPE_CLASS.TYPE_DWORD:
		pDWORD := value.pValue;
		wsString := WCONCAT(wsString, TO_WSTRING(pDWORD^));
		
	__SYSTEM.TYPE_CLASS.TYPE_LWORD:
		pLWORD := value.pValue;
		wsString := WCONCAT(wsString, TO_WSTRING(pLWORD^));
		
	__SYSTEM.TYPE_CLASS.TYPE_SINT:
		pSINT := value.pValue;
		wsString := WCONCAT(wsString, TO_WSTRING(pSINT^));
		
	__SYSTEM.TYPE_CLASS.TYPE_INT:
		pINT := value.pValue;
		wsString := WCONCAT(wsString, TO_WSTRING(pINT^));
		
	__SYSTEM.TYPE_CLASS.TYPE_DINT:
		pDINT := value.pValue;
		wsString := WCONCAT(wsString, TO_WSTRING(pDINT^));
		
	__SYSTEM.TYPE_CLASS.TYPE_LINT:
		pLINT := value.pValue;
		wsString := WCONCAT(wsString, TO_WSTRING(pLINT^));
		
	__SYSTEM.TYPE_CLASS.TYPE_USINT:
		pUSINT := value.pValue;
		wsString := WCONCAT(wsString, TO_WSTRING(pUSINT^));
		
	__SYSTEM.TYPE_CLASS.TYPE_UINT:
		pUINT := value.pValue;
		wsString := WCONCAT(wsString, TO_WSTRING(pUINT^));
		
	__SYSTEM.TYPE_CLASS.TYPE_UDINT:
		pUDINT := value.pValue;
		wsString := WCONCAT(wsString, TO_WSTRING(pUDINT^));
		
	__SYSTEM.TYPE_CLASS.TYPE_ULINT:
		pULINT := value.pValue;
		wsString := WCONCAT(wsString, TO_WSTRING(pULINT^));
		
	__SYSTEM.TYPE_CLASS.TYPE_REAL:
		pREAL := value.pValue;
		wsString := WCONCAT(wsString, TO_WSTRING(pREAL^));
		
	__SYSTEM.TYPE_CLASS.TYPE_LREAL:
		pLREAL := value.pValue;
		wsString := WCONCAT(wsString, TO_WSTRING(pLREAL^));
		
	__SYSTEM.TYPE_CLASS.TYPE_TIME:
		pTIME := value.pValue;
		wsString := WCONCAT(wsString, TO_WSTRING(pTIME^));
		
	__SYSTEM.TYPE_CLASS.TYPE_LTIME:
		pLTIME := value.pValue;
		wsString := WCONCAT(wsString, TO_WSTRING(pLTIME^));
	
	__SYSTEM.TYPE_CLASS.TYPE_DATE:
		pDATE := value.pValue;
		wsString := WCONCAT(wsString, TO_WSTRING(pDATE^));
		
	__SYSTEM.TYPE_CLASS.TYPE_DATEANDTIME:
		pDT := value.pValue;
		wsString := WCONCAT(wsString, TO_WSTRING(pDT^));
		
	__SYSTEM.TYPE_CLASS.TYPE_TIMEOFDAY:
		pTOD := value.pValue;
		wsString := WCONCAT(wsString, TO_WSTRING(pTOD^));
		
	__SYSTEM.TYPE_CLASS.TYPE_ENUM: // does not work!
		pENUM := value.pValue;
		wsString := WCONCAT(wsString, TO_WSTRING(pENUM^));

END_CASE

AppendAny := THIS^;
END_METHOD

METHOD PUBLIC Clear : I_WStringBuilder // Clear the current build string.
VAR_INPUT
END_VAR
wsString := "";
Clear := THIS^;
END_METHOD

METHOD PUBLIC Insert : I_WStringBuilder
VAR_INPUT
	text	 : WSTRING;	// Text to append to current build string
	position : INT;		// Insert position (Index)
END_VAR
wsString := Tc2_Standard.WINSERT(wsString, text, position);
Insert := THIS^;
END_METHOD

METHOD PUBLIC Reset : I_WStringBuilder //Reset current build string to an empty string.
VAR_INPUT
END_VAR
wsString := "";
Reset := THIS^;
END_METHOD

METHOD PUBLIC Set : I_WStringBuilder
VAR_INPUT
	text : WSTRING; //Text to append to current build string
END_VAR
wsString := text;
Set := THIS^;
END_METHOD

METHOD PUBLIC ToString : T_MaxString // Returns current build string.
VAR
	str	  : T_MaxString;
END_VAR
WSTRING_TO_STRING2(ADR(str), ADR(wsString), SIZEOF(str));
ToString := str;
END_METHOD

METHOD PUBLIC ToWString : WSTRING // Returns current build string.
VAR_INPUT
END_VAR
ToWString := wsString;
END_METHOD

END_FUNCTION_BLOCK

// ---- POUs/Components/_Base/FB_ManualUiBase.TcPOU
FUNCTION_BLOCK PUBLIC ABSTRACT FB_ManualUiBase IMPLEMENTS I_ManualUi
VAR_INPUT
	// object name
	stName 					: ST_Text;
	// objekts index
	diObjectIndex			: DINT;
	// selected object index in hmi 
	diSelectedObjectIndex	: DINT;
	/// manual mode enable
	bEnableManual			: BOOL;
	/// device BMK
	stBmk					: ST_Text;
	// state object
	stStateObject			: REFERENCE TO ST_Object_Item;
END_VAR
VAR_OUTPUT
	/// Fehler
	bError				: BOOL;
	/// Fehlertext
	stErrorText			: ST_Text;
	/// Warnung
	bWarning			: BOOL;
	/// Warnungstext
	stWarnText			: ST_Text;
END_VAR
VAR
	bManualActive			: BOOL;
END_VAR

// to be subclassed..

METHOD M_SetStateObject : BOOL
VAR_IN_OUT
	stStateObjectRef	: ST_Object_Item;
END_VAR
stStateObject REF= stStateObjectRef;
END_METHOD

PROPERTY Name : ST_Text
GET
Name := stName;
END_GET
END_PROPERTY

PROPERTY ObjectIndex : DINT
GET
ObjectIndex := diObjectIndex;
END_GET
SET
diObjectIndex := ObjectIndex;
END_SET
END_PROPERTY

END_FUNCTION_BLOCK

// ---- POUs/System/Utilities/String/WConcat3.TcPOU
FUNCTION WConcat3 : WSTRING(255)
VAR_INPUT
	wsExpression1: WSTRING(255);
	wsExpression2: WSTRING(255);
	wsExpression3: WSTRING(255);
END_VAR

WConcat3 := WCONCAT(wsExpression1, wsExpression2);
WConcat3 := WCONCAT(WConcat3, wsExpression3);

END_FUNCTION

// ---- POUs/Components/AxisDriver/FB_AxisDriver.TcPOU
/// Axis driver function block
FUNCTION_BLOCK FB_AxisDriver EXTENDS FB_ComponentBase IMPLEMENTS ITFMotionComponent
VAR_INPUT
	/// AmsNetId of the IPC 
	IPCNetID		: T_AmsNetId := '';
	/// Auto Disable Funktion
	bEnableAutoPowerOff : BOOL := FALSE;
	/// Drehmomentfaktor
	fTorqueFactor 	: REAL := 1;
	
	// axis prm
	stDefaultPrm	: ST_AxisDriverParameter;
	stHomingPrm		: ST_AxisHomingParameter;
	
	// enable inputs
	bEnable			: BOOL;
	bEnableNeg 		: BOOL;
	bEnablePos 		: BOOL;
	bCalibrationCam	: BOOL;
	
	bAX5805_Error	: BOOL;		(*	AX5805 Fehler liegt an - Safety Reset erforderlich	*)
	
	tEnableTime		: TIME := T#1000MS;	
END_VAR
VAR_OUTPUT
	/// Fehlerzustand
	bError				:BOOL;
	/// Fehlertext
	stErrorText			:ST_Text;
	/// Fehlertext Zusatz
	stErrorText_Add		:ST_Text;
	/// Warnung
	bWarning			:BOOL;
	/// Warnungstext
	stWarnText			:ST_Text;
		
	/// Achse aktiv
	Operational: BOOL;
	/// Position der Achse
	Position: LREAL;
	///Aktuelle Modulo Position
	ModuloPosition: LREAL;
	/// Aktuelle Positionen mit gelatchten Objektposition gleich
	bLatchedObjPositionOK					:BOOL;
	/// Schleppfehler
	fPosDiff								:LREAL;
	/// Axis is Homed
	Homed									:BOOL;
	
	/// Position offset set
	bSetPositionOffsetDone					:BOOL;
	/// Current position offset value
	fCurrentPositionOffset					:LREAL;
	///has job
	bHasJob									: BOOL;
	bHoldActiv								: BOOL;
	// move abs is ready
	bMovAbsRdy								: BOOL; 
END_VAR
VAR
	/// Axis ID and reference
	eAxisId: E_Axis;
	fbAxisRef: REFERENCE TO AXIS_REF;
	/// Additional (direct) linked inputs
	stIn: REFERENCE TO ST_AxisIn;
	/// Additional (direct) linked outputs
	stOut: REFERENCE TO ST_AxisOut;
	///	AX5000 - axes diag + reset 
	fbAX5xxxDiag: FB_AX5000Diag;
	stAX5xxxDiag: ST_AX5000Diag;
	/// Indradrive  - axes diag + reset 
	fbIndraDrvDiag: FB_IndraDriveDiag;
	stIndraDrvDiag: ST_IndraDriveDiag;
	/// Device ref: contains sNetID of EcMaster, nSlaveAddr of EcDrive, nDriveNo of EcDrive, either preset or read from NC 
	stDriveRef: ST_DriveRef;
	/// FB for axis enabling
	fbPower: MC_Power;
	/// FB for halting the axis
	fbHalt: MC_Halt;
	stHaltPrm: ST_AxisHaltParameter;
	/// FB for stopping the axis
	fbStop: MC_Stop;
	stStopPrm: ST_AxisStopParameter;
	/// FB for resetting the axis
	fbReset: MC_Reset;
	/// FB for axis homing
	fbHoming: MC_Home;	
	/// FB for set axis position
	fbSetPos: MC_SetPosition;
	stSetPosPrm: ST_AxisSetPosParameter;
	/// FB for set axis AX5000 position offset
	fbAxSetPosOffs: FB_SoEAX5000SetPositionOffset;
	/// FB for axis jog
	fbjog: MC_Jog;
	stJogPrm: ST_AxisJogParameter;
	/// FB for axis accelerating jog
	fbJogAcc: MC_MoveVelocity;
	stJogAccPrm: ST_AxisJogAccParameter;
	tonJogAcc: TON;
	/// FB for axis move absolute (this motion command can be overlayed, thus 2 FBs)
	fbMovAbs1: MC_MoveAbsolute;
	fbMovAbs2: MC_MoveAbsolute;
	stMovAbsPrm: ST_AxisMoveAbsParameter;
	/// FB for axis move additive (this motion command can be overlayed, thus 2 FBs)
	fbMovAdd1: MC_MoveAdditive;
	fbMovAdd2: MC_MoveAdditive;
	stMovAddPrm: ST_AxisMoveAddParameter;
	/// FB for axis move relative (this motion command can be overlayed, thus 2 FBs)
	fbMovRel1: MC_MoveRelative;
	fbMovRel2: MC_MoveRelative;
	stMovRelPrm: ST_AxisMoveRelParameter;
	/// FB for axis move modulo (this motion command can be overlayed, thus 2 FBs)
	fbMovMod1: MC_MoveModulo;
	fbMovMod2: MC_MoveModulo;
	stMovModPrm: ST_AxisMoveModParameter;
	/// FB for axis move velocity (this motion command can be overlayed, thus 2 FBs)
	fbMovVel1: MC_MoveVelocity;
	fbMovVel2: MC_MoveVelocity;
	stMovVelPrm: ST_AxisMoveVelParameter;
	/// FB for axis dynamic gear
	fbGearIn: MC_GearInDyn;
	stGearInPrm: ST_AxisGearInParameter;
	fbGearOut: MC_GearOut;
	stGearOutPrm: ST_AxisGearOutParameter;
	/// FB for axis torque control
	fbTorqueControl: MC_TorqueControl;
	stTorqCtrlPrm: ST_AxisTorqCtrlParameter;
	/// private workflow var`s	
	eMasterAxisId: E_Axis;
	eAxisType: E_AxisType;	
	/// requested motion command
	eCommandRequest: E_MotionCommand;
	/// actual motion command
	eCommandExecute: E_MotionCommand;
	///tonTimeOut	: TON;
	nErrorID: UDINT;
	rtrigError: R_TRIG;
	ftrigDiag: F_TRIG;
	ftrigDiagIndradrv: F_TRIG;
	bErrDiagActive: BOOL;
	tonChkOperation: TON;
	sMsg: T_MaxString;
	//ii: INT;
	/// ID of the last error in one of the motion FBs
	tonAutoPowerOff: TON;
	tonEnable	:TON;
	posPowerError	:R_TRIG;
	fPosLatched	:LREAL;
	//timeout positioning
	tonTimeout: TON;
	
	// SoE	
	stSoE	: ST_AxisSoE;
	diTempVal	:DINT;
	
	bStartInitPosOffset		:BOOL;
	fPosOffsetValToSet		:LREAL;
	
	bHold					: BOOL;
	fSetOverride			: LREAL := 100.0;	
END_VAR

///
/// Axis driver FB
/// TP/www.rmth.at/2014
/// RE/2021 - 	Extend AX5000 Diagnostic
///				Add InitPositionOffset
/// 

Run();

/// Actual amplifier temp. [°C]
{attribute 'monitoring' := 'call'}
PROPERTY AmplifierTemp : LREAL
GET
/// Actual amplifier temp. [°C]
AmplifierTemp := INT_TO_LREAL(stIn.iAmplifierTemperature) / 10;
END_GET
END_PROPERTY

/// Get's the axis reference
PROPERTY Axis : AXIS_REF
GET
Axis := fbAxisRef;
END_GET
END_PROPERTY

{attribute 'monitoring' := 'call'}
PROPERTY AxisId : E_Axis
GET
AxisId := eAxisId;
END_GET
SET
eAxisId := AxisId;
END_SET
END_PROPERTY

/// Get`s the MC axis state.
PROPERTY AxisState : Tc2_MC2.ST_AxisStatus
GET
AxisState := fbAxisRef.Status;
END_GET
END_PROPERTY

{attribute 'monitoring' := 'call'}
PROPERTY AxisType : E_AxisType
GET
AxisType := eAxisType;
END_GET
SET
eAxisType := AxisType;
END_SET
END_PROPERTY

ACTION CheckLatchState:
bLatchedObjPositionOK := ABS(Position - fPosLatched) <= 0.1;
END_ACTION

/// Coupled (Slave) Info
{attribute 'monitoring' := 'call'}
PROPERTY Coupled : BOOL
GET
Coupled := fbAxisRef.Status.Coupled;
END_GET
END_PROPERTY

PROPERTY DefaultParameter : ST_AxisDriverParameter
GET
DefaultParameter := stDefaultPrm;
END_GET
SET
stDefaultPrm := DefaultParameter;
END_SET
END_PROPERTY

{attribute 'monitoring' := 'call'}
PROPERTY Enable : BOOL
GET
Enable := bEnable;
END_GET
SET
bEnable := Enable;
END_SET
END_PROPERTY

{attribute 'monitoring' := 'call'}
PROPERTY EnableNeg : BOOL
GET
EnableNeg:=bEnableNeg;
END_GET
SET
bEnableNeg:=EnableNeg;
END_SET
END_PROPERTY

{attribute 'monitoring' := 'call'}
PROPERTY EnablePos : BOOL
GET
EnablePos := bEnablePos;
END_GET
SET
bEnablePos := EnablePos;
END_SET
END_PROPERTY

/// Performs an electronic axis gear-in using default parameter set.
{attribute 'object_name' := 'GearIn'}
METHOD GearIn : E_OperationResult
VAR_INPUT
	/// Gear ratio
	fRatio: LREAL;
	/// Master axis id
	eMasterId: E_Axis;
END_VAR
VAR_IN_OUT
	/// Master axis to gear-in to
	fbMaster: AXIS_REF;
END_VAR
// gear in axis to master

// init result pessimistic
GearIn := E_OperationResult.eOperationResult_NOk;

// if stopping or resetting is active return --> higher prio
IF eCommandExecute = E_MotionCommand.eMotionCommand_reset OR eCommandExecute = E_MotionCommand.eMotionCommand_stop THEN
	RETURN;
END_IF

stGearInPrm := stDefaultPrm.stGearInPrm;
stGearInPrm.fGearRatio := fRatio;
stGearInPrm.eMasterId := eMasterId;
stGearInPrm.fbMaster REF= fbMaster;

eCommandRequest := E_MotionCommand.eMotionCommand_gearIn;
GearIn := E_OperationResult.eOperationResult_Ok;
END_METHOD

/// Performs an electronic axis gear-in using specified parameter
{attribute 'object_name' := 'GearInEx'}
METHOD GearInEx : E_OperationResult
VAR_IN_OUT
	/// Parameter set to use
	stGearInParameter: ST_AxisGearInParameter;
END_VAR
// gear in axis to master

GearInEx := THIS^.GearIn(stGearInParameter.fGearRatio, stGearInParameter.eMasterId, stGearInParameter.fbMaster);

IF GearInEx = E_OperationResult.eOperationResult_Ok THEN
	stGearInPrm := stGearInParameter;
END_IF
END_METHOD

/// Performs an electronic axis gear-out using default parameter set.
{attribute 'object_name' := 'GearOut'}
METHOD GearOut : E_OperationResult
// gear out axis from master

// init result pessimistic
GearOut := E_OperationResult.eOperationResult_NOk;

// if stopping is active return --> higher prio
IF eCommandExecute = E_MotionCommand.eMotionCommand_stop THEN
	RETURN;
END_IF

stGearOutPrm := stDefaultPrm.stGearOutPrm;
eCommandRequest := E_MotionCommand.eMotionCommand_gearOut;
GearOut := E_OperationResult.eOperationResult_Ok;
END_METHOD

/// Performs an electronic axis gear-out using specified parameter
{attribute 'object_name' := 'GearOutEx'}
METHOD GearOutEx : E_OperationResult
VAR_IN_OUT
	/// Parameter set to use
	stGearOutParameter: ST_AxisGearOutParameter;
END_VAR
// gear in axis to master

GearOutEx := THIS^.GearOut();

IF GearOutEx = E_OperationResult.eOperationResult_Ok THEN
	stGearOutPrm := stGearOutParameter;
END_IF
END_METHOD

/// Get's or set's the gear ratio for MC_GearInDyn.
{attribute 'monitoring' := 'call'}
PROPERTY GearRatio : LREAL
GET
// return actual gear ratio
GearRatio := stGearInPrm.fGearRatio;
END_GET
SET
// Updates the gear-ratio (only effective if GearIn was called bevore).
stGearInPrm.fGearRatio := GearRatio;
END_SET
END_PROPERTY

/// Axis halt using default parameter
{attribute 'object_name' := 'Halt'}
METHOD Halt : E_OperationResult
// halt axis

// init result pessimistic
Halt := E_OperationResult.eOperationResult_NOk;

// if stopping is active return --> higher prio: stop
IF eCommandExecute = E_MotionCommand.eMotionCommand_stop THEN
	RETURN;
END_IF

stHaltPrm := stDefaultPrm.stHaltPrm;
//ILog.AddLog('Request received: halt', Concat2('AxisDriver', INT_TO_STRING(THIS^.ID)), E_LogLevel.eLogLevelInformation);
eCommandRequest := E_MotionCommand.eMotionCommand_halt;
Halt := E_OperationResult.eOperationResult_Ok;
// sofort aufrufen
Run();
END_METHOD

/// Axis halt using specified parameter
{attribute 'object_name' := 'HaltEx'}
METHOD HaltEx : E_OperationResult
VAR_INPUT
	/// Parameter set to use
	stHaltParameter: ST_AxisHaltParameter;
END_VAR
// halt axis

HaltEx := THIS^.Halt();

IF HaltEx = E_OperationResult.eOperationResult_Ok THEN
	stHaltPrm := stHaltParameter;
END_IF
END_METHOD

METHOD PUBLIC Hold : BOOL
VAR_INPUT
END_VAR
bHold := true;
END_METHOD

/// Axis home using default parameter
{attribute 'object_name' := 'Home'}
METHOD Home : E_OperationResult
// home axis

// init result pessimistic
Home := E_OperationResult.eOperationResult_NOk;

// if stopping or resetting is active return --> higher prio
IF eCommandExecute = E_MotionCommand.eMotionCommand_reset OR eCommandExecute = E_MotionCommand.eMotionCommand_stop THEN
	RETURN;
END_IF

stHomingPrm := stDefaultPrm.stHomingPrm;

eCommandRequest := E_MotionCommand.eMotionCommand_home;
Home := E_OperationResult.eOperationResult_Ok;
END_METHOD

/// Axis home using specified parameter
{attribute 'object_name' := 'HomeEx'}
METHOD HomeEx : E_OperationResult
VAR_INPUT
	/// Parameter set to use
	stHomingParameter: ST_AxisHomingParameter;
END_VAR
// home axis

HomeEx := THIS^.Home();

IF HomeEx = E_OperationResult.eOperationResult_Ok THEN
	stHomingPrm := stHomingParameter;
END_IF
END_METHOD

METHOD PUBLIC InitPosOffset : BOOL
VAR_INPUT
	fPositionOffset				:LREAL;
END_VAR
// check ready
IF bStartInitPosOffset THEN
	InitPosOffset := FALSE;
	RETURN;
END_IF

bStartInitPosOffset	:= TRUE;
fPosOffsetValToSet := fPositionOffset;
END_METHOD

/// Gets the InTorque output for TorqueControl.
{attribute 'monitoring' := 'call'}
PROPERTY PUBLIC InTorque : BOOL
GET
InTorque := fbTorqueControl.InTorque;
END_GET
END_PROPERTY

/// Axis jog using default parameter
/// This method must be called cyclic (otherwise jog Fwd/Bwd will be reset)
{attribute 'object_name' := 'Jog'}
METHOD Jog : E_OperationResult
VAR_INPUT
	bJogBackwards: BOOL;
	bJogForward: BOOL;
END_VAR
// jog axis

// init result pessimistic
Jog := E_OperationResult.eOperationResult_NOk;

// if stopping or resetting is active return --> higher prio
IF eCommandExecute = E_MotionCommand.eMotionCommand_reset OR eCommandExecute = E_MotionCommand.eMotionCommand_stop THEN
	RETURN;
END_IF

stJogPrm := stDefaultPrm.stJogPrm;
stJogPrm.bJogBackwards := bJogBackwards;
stJogPrm.bJogForward := bJogForward;

IF stJogPrm.bJogBackwards OR stJogPrm.bJogForward THEN
	eCommandRequest := E_MotionCommand.eMotionCommand_jog;
END_IF

Jog := E_OperationResult.eOperationResult_Ok;
END_METHOD

/// Axis jog accelerating using default parameter
/// This method must be called cyclic (otherwise jog Fwd/Bwd will be reset)
{attribute 'object_name' := 'JogAcc'}
METHOD JogAcc : E_OperationResult
VAR_INPUT
	bJogBackwards: BOOL;
	bJogForward: BOOL;
END_VAR
// jog axis acc

// init result pessimistic
JogAcc := E_OperationResult.eOperationResult_NOk;

// if stopping or resetting is active return --> higher prio
IF eCommandExecute = E_MotionCommand.eMotionCommand_reset OR eCommandExecute = E_MotionCommand.eMotionCommand_stop THEN
	RETURN;
END_IF

stJogAccPrm := stDefaultPrm.stJogAccPrm;
stJogAccPrm.bJogBackwards := bJogBackwards;
stJogAccPrm.bJogForward := bJogForward;

IF stJogAccPrm.bJogBackwards OR stJogAccPrm.bJogForward THEN
	eCommandRequest := E_MotionCommand.eMotionCommand_jogAcc;
END_IF

JogAcc := E_OperationResult.eOperationResult_Ok;
END_METHOD

/// Axis jog accelerating using specified parameter
{attribute 'object_name' := 'JogAccEx'}
METHOD JogAccEx : E_OperationResult
VAR_INPUT
	/// Parameter set to use
	stJogAccParameter: ST_AxisJogAccParameter;
END_VAR
// jog acc axis

JogAccEx := THIS^.JogAcc(stJogAccParameter.bJogBackwards, stJogAccParameter.bJogForward);

IF JogAccEx = E_OperationResult.eOperationResult_Ok THEN
	stJogAccPrm := stJogAccParameter;
END_IF
END_METHOD

/// Axis jog accelerating using default parameter
/// This method must be called cyclic (otherwise jog Fwd/Bwd will be reset)
{attribute 'object_name' := 'JogAccExVel'}
METHOD JogAccExVel : E_OperationResult
VAR_INPUT
	bJogBackwards: BOOL;
	bJogForward: BOOL;
	/// Slow (starting) speed
	fSlowSpeed: LREAL;
	/// Fast end-speed
	fFastSpeed: LREAL;
	/// Time for ramp from slow to fast speed [ms]
	fAccTime: LREAL;
END_VAR
// jog axis acc

// init result pessimistic
JogAccExVel := E_OperationResult.eOperationResult_NOk;

// if stopping or resetting is active return --> higher prio
IF eCommandExecute = E_MotionCommand.eMotionCommand_reset OR eCommandExecute = E_MotionCommand.eMotionCommand_stop THEN
	RETURN;
END_IF

stJogAccPrm := stDefaultPrm.stJogAccPrm;
stJogAccPrm.fSlowSpeed := fSlowSpeed;
stJogAccPrm.fFastSpeed := fFastSpeed;
stJogAccPrm.tAccTime := LREAL_TO_TIME(fAccTime);
stJogAccPrm.bJogBackwards := bJogBackwards;
stJogAccPrm.bJogForward := bJogForward;

IF stJogAccPrm.bJogBackwards OR stJogAccPrm.bJogForward THEN
	eCommandRequest := E_MotionCommand.eMotionCommand_jogAcc;
END_IF

JogAccExVel := E_OperationResult.eOperationResult_Ok;
END_METHOD

/// Axis jog using specified parameter
{attribute 'object_name' := 'JogEx'}
METHOD JogEx : E_OperationResult
VAR_INPUT
	/// Parameter set to use
	stJogParameter: ST_AxisJogParameter;
END_VAR
// jog axis

JogEx := THIS^.Jog(stJogParameter.bJogBackwards, stJogParameter.bJogForward);

IF JogEx = E_OperationResult.eOperationResult_Ok THEN
	stJogPrm := stJogParameter;
END_IF
END_METHOD

/// Axis jog using specified parameter
METHOD JogExVel : E_OperationResult
VAR_INPUT
	bJogBackwards 	: BOOL;
	bJogForward		: BOOL;
	/// Velocity
	fVelocity		: LREAL;
	/// Modus
	eMode: E_JogMode := E_JogMode.MC_JOGMODE_INCHING;
END_VAR
// jog axis

JogExVel := THIS^.Jog(bJogBackwards, bJogForward);

IF JogExVel = E_OperationResult.eOperationResult_Ok THEN
	stJogPrm := stDefaultPrm.stJogPrm;
	stJogPrm.eMode := eMode;
	stJogPrm.fVelocity := fVelocity;
	stJogPrm.bJogBackwards := bJogBackwards;
	stJogPrm.bJogForward := bJogForward;
END_IF
END_METHOD

{attribute 'monitoring' := 'call'}
PROPERTY LastMcErrorId : UDINT
GET
LastMcErrorId := nErrorID;
END_GET
END_PROPERTY

METHOD LatchObjState : BOOL
VAR_INPUT
END_VAR
fPosLatched := Position;
END_METHOD

METHOD PRIVATE M_SetLocalError : BOOL
VAR_INPUT
	stErrorText1		: ST_Text;
END_VAR
eState := E_ComponentState.eComponentState_error;
stErrorText := stErrorText1;
sLastError := TO_STRING(stErrorText1.wsName);
END_METHOD

METHOD PRIVATE M_SetLocalErrorEx : BOOL
VAR_INPUT
	stErrorText1		: ST_Text;
	stErrorTextAdd		: ST_Text;
END_VAR
eState := E_ComponentState.eComponentState_error;
stErrorText := stErrorText1;
stErrorText_Add := stErrorTextAdd;
sLastError := TO_STRING(stErrorText1.wsName);
END_METHOD

METHOD PRIVATE M_SetLocalErrorS : BOOL
VAR_INPUT
	sErrorText1		: STRING;
	sErrorText2		: STRING;
END_VAR
VAR
	stErrorText		: ST_Text;
END_VAR
eState := E_ComponentState.eComponentState_error;

stErrorText := F_CreateDynText(TO_WSTRING(CONCAT(sErrorText1, sErrorText2)), 0);
sLastError := TO_STRING(stErrorText.wsName);
END_METHOD

{attribute 'monitoring' := 'call'}
PROPERTY MasterAxisId : E_Axis
GET
MasterAxisId := eMasterAxisId;
END_GET
END_PROPERTY

/// Get's a value, indicating whether axis position is within motulo target position window and not moving.
/// Position window: default epsilon (1E-3).
/// Valid for previous MOD movement's.
METHOD PUBLIC ModuloReached : BOOL
VAR_INPUT
END_VAR
ModuloReached := ModuloWindowReached(fEpsilon);
END_METHOD

/// Get's a value, indicating whether axis position is within modulo target position window and not moving.
/// Valid for previous MOD movement's. 
METHOD PUBLIC ModuloWindowReached : BOOL
VAR_INPUT
	fWindow : LREAL;
END_VAR
ModuloWindowReached := ModuloPosition >= (stMovModPrm.fPosition - fWindow) AND ModuloPosition <= (stMovModPrm.fPosition + fWindow) AND NotMoving;
END_METHOD

/// Actual motor temp. [°C]
{attribute 'monitoring' := 'call'}
PROPERTY MotorTemp : LREAL
GET
/// Actual motor temp. [°C]
MotorTemp := INT_TO_LREAL(stIn.iMotorTemperature) / 10;
END_GET
END_PROPERTY

/// Performs an absolute axis positioning using default parameter set.
/// This motion is capable to overlay (max. 2 parallel at one time)
{attribute 'object_name' := 'MoveAbs'}
METHOD MoveAbs : E_OperationResult
VAR_INPUT
	/// Position to move to
	fPosition: LREAL;
END_VAR
// move axis abs

// init result pessimistic
MoveAbs := E_OperationResult.eOperationResult_NOk;

// if stopping or resetting is active return --> higher prio
IF eCommandExecute = E_MotionCommand.eMotionCommand_reset OR eCommandExecute = E_MotionCommand.eMotionCommand_stop THEN
	RETURN;
END_IF

stMovAbsPrm := stDefaultPrm.stMovAbsPrm;
stMovAbsPrm.fPosition := fPosition;

eCommandRequest := E_MotionCommand.eMotionCommand_moveAbs;
MoveAbs := E_OperationResult.eOperationResult_Ok;
END_METHOD

/// Performs an absolute axis positioning using input parameter set.
/// This motion is capable to overlay (max. 2 parallel at one time)
{attribute 'object_name' := 'MoveAbsAccDec'}
METHOD MoveAbsAccDec : E_OperationResult
VAR_INPUT
	/// Position to move to
	fPosition: LREAL;
	/// Speed
	fVelocity: LREAL;
	/// Acceleration
	fAcceleration	: LREAL;
	/// Deceleration
	fDeceleration	: LREAL;
END_VAR
// move axis abs

// init result pessimistic
MoveAbsAccDec := E_OperationResult.eOperationResult_NOk;

// if stopping or resetting is active return --> higher prio
IF eCommandExecute = E_MotionCommand.eMotionCommand_reset OR eCommandExecute = E_MotionCommand.eMotionCommand_stop THEN
	RETURN;
END_IF

stMovAbsPrm := stDefaultPrm.stMovAbsPrm;
stMovAbsPrm.fPosition := fPosition;
stMovAbsPrm.fVelocity := fVelocity;
stMovAbsPrm.fAcceleration := fAcceleration;
stMovAbsPrm.fDeceleration := fDeceleration;

eCommandRequest := E_MotionCommand.eMotionCommand_moveAbs;
MoveAbsAccDec := E_OperationResult.eOperationResult_Ok;
END_METHOD

/// Performs an absolute axis positioning using specified parameter
/// This motion is capable to overlay (max. 2 parallel at one time)
{attribute 'object_name' := 'MoveAbsEx'}
METHOD MoveAbsEx : E_OperationResult
VAR_INPUT
	/// Parameter set to use
	stMovAbsParameter: ST_AxisMoveAbsParameter;
END_VAR
// move axis abs

MoveAbsEx := THIS^.MoveAbs(stMovAbsParameter.fPosition);

IF MoveAbsEx = E_OperationResult.eOperationResult_Ok THEN
	stMovAbsPrm := stMovAbsParameter;
END_IF
END_METHOD

/// Performs an absolute axis positioning using input parameter set.
/// This motion is capable to overlay (max. 2 parallel at one time)
{attribute 'object_name' := 'MoveAbsExVel'}
METHOD MoveAbsExVel : E_OperationResult
VAR_INPUT
	/// Position to move to
	fPosition		: LREAL;
	/// Speed
	fVelocity		: LREAL;
END_VAR
// move axis abs

// init result pessimistic
MoveAbsExVel := E_OperationResult.eOperationResult_NOk;

// if stopping or resetting is active return --> higher prio
IF eCommandExecute = E_MotionCommand.eMotionCommand_reset OR eCommandExecute = E_MotionCommand.eMotionCommand_stop THEN
	RETURN;
END_IF

stMovAbsPrm := stDefaultPrm.stMovAbsPrm;
stMovAbsPrm.fPosition := fPosition;
stMovAbsPrm.fVelocity := fVelocity;

eCommandRequest := E_MotionCommand.eMotionCommand_moveAbs;
MoveAbsExVel := E_OperationResult.eOperationResult_Ok;
END_METHOD

/// Performs an additive axis positioning using default parameter set.
/// This motion is capable to overlay (max. 2 parallel at one time)
{attribute 'object_name' := 'MoveAdd'}
METHOD MoveAdd : E_OperationResult
VAR_INPUT
	/// Distance
	fDistance: LREAL;
END_VAR
// move axis add

// init result pessimistic
MoveAdd := E_OperationResult.eOperationResult_NOk;

// if stopping or resetting is active return --> higher prio
IF eCommandExecute = E_MotionCommand.eMotionCommand_reset OR eCommandExecute = E_MotionCommand.eMotionCommand_stop THEN
	RETURN;
END_IF

stMovAddPrm := stDefaultPrm.stMovAddPrm;
stMovAddPrm.fDistance := fDistance;

eCommandRequest := E_MotionCommand.eMotionCommand_moveAdd;
MoveAdd := E_OperationResult.eOperationResult_Ok;
END_METHOD

/// Performs an additive axis positioning using specified parameter set.
/// This motion is capable to overlay (max. 2 parallel at one time)
{attribute 'object_name' := 'MoveAddEx'}
METHOD MoveAddEx : E_OperationResult
VAR_INPUT
	/// Parameter set to use
	stMovAddParameter: ST_AxisMoveAddParameter;
END_VAR
// move axis add

MoveAddEx := THIS^.MoveAdd(stMovAddParameter.fDistance);

IF MoveAddEx = E_OperationResult.eOperationResult_Ok THEN
	stMovAddPrm := stMovAddParameter;
END_IF
END_METHOD

/// Performs an modulo axis positioning using default parameter set.
/// This motion is capable to overlay (max. 2 parallel at one time)
{attribute 'object_name' := 'MoveMod'}
METHOD MoveMod : E_OperationResult
VAR_INPUT
	/// Position to move to
	fPosition: LREAL;
END_VAR
// move axis mod

// init result pessimistic
MoveMod := E_OperationResult.eOperationResult_NOk;

// if stopping or resetting is active return --> higher prio
IF eCommandExecute = E_MotionCommand.eMotionCommand_reset OR eCommandExecute = E_MotionCommand.eMotionCommand_stop THEN
	RETURN;
END_IF

stMovModPrm := stDefaultPrm.stMovModPrm;
stMovModPrm.fPosition := fPosition;

eCommandRequest := E_MotionCommand.eMotionCommand_moveMod;
MoveMod := E_OperationResult.eOperationResult_Ok;
END_METHOD

/// Performs an modulo axis positioning using specified parameter
/// This motion is capable to overlay (max. 2 parallel at one time)
{attribute 'object_name' := 'MoveModEx'}
METHOD MoveModEx : E_OperationResult
VAR_INPUT
	/// Parameter set to use
	stMovModParameter: ST_AxisMoveModParameter;
END_VAR
// move axis mod

MoveModEx := THIS^.MoveMod(stMovModParameter.fPosition);

IF MoveModEx = E_OperationResult.eOperationResult_Ok THEN
	stMovModPrm := stMovModParameter;
END_IF
END_METHOD

/// Performs an modulo axis positioning using input parameter set.
/// This motion is capable to overlay (max. 2 parallel at one time)
{attribute 'object_name' := 'MoveModExVel'}
METHOD MoveModExVel : E_OperationResult
VAR_INPUT
	/// Position to move to
	fPosition: LREAL;
	/// Speed
	fVelocity: LREAL;
END_VAR
// move axis abs

// init result pessimistic
MoveModExVel := E_OperationResult.eOperationResult_NOk;

// if stopping or resetting is active return --> higher prio
IF eCommandExecute = E_MotionCommand.eMotionCommand_reset OR eCommandExecute = E_MotionCommand.eMotionCommand_stop THEN
	RETURN;
END_IF

stMovModPrm := stDefaultPrm.stMovModPrm;
stMovModPrm.fPosition := fPosition;
stMovModPrm.fVelocity := fVelocity;

eCommandRequest := E_MotionCommand.eMotionCommand_moveMod;
MoveModExVel := E_OperationResult.eOperationResult_Ok;
END_METHOD

/// Performs an relative axis positioning using default parameter set.
/// This motion is capable to overlay (max. 2 parallel at one time)
{attribute 'object_name' := 'MoveRel'}
METHOD MoveRel : E_OperationResult
VAR_INPUT
	/// Distance
	fDistance: LREAL;
END_VAR
// move axis rel

// init result pessimistic
MoveRel := E_OperationResult.eOperationResult_NOk;

// if stopping or resetting is active return --> higher prio
IF eCommandExecute = E_MotionCommand.eMotionCommand_reset OR eCommandExecute = E_MotionCommand.eMotionCommand_stop THEN
	RETURN;
END_IF

stMovRelPrm := stDefaultPrm.stMovRelPrm;
stMovRelPrm.fDistance := fDistance;

eCommandRequest := E_MotionCommand.eMotionCommand_moveRel;
MoveRel := E_OperationResult.eOperationResult_Ok;
END_METHOD

/// Performs an relative axis positioning using specified parameter set.
/// This motion is capable to overlay (max. 2 parallel at one time)
{attribute 'object_name' := 'MoveRelAccDec'}
METHOD MoveRelAccDec : E_OperationResult
VAR_INPUT
	/// Distance to move to
	fDistance: LREAL;
	/// Speed
	fVelocity: LREAL;
	/// Acceleration
	fAcceleration	: LREAL;
	/// Deceleration
	fDeceleration	: LREAL;
END_VAR
// move axis rel

// init result pessimistic
MoveRelAccDec := E_OperationResult.eOperationResult_NOk;

// if stopping or resetting is active return --> higher prio
IF eCommandExecute = E_MotionCommand.eMotionCommand_reset OR eCommandExecute = E_MotionCommand.eMotionCommand_stop THEN
	RETURN;
END_IF

stMovRelPrm := stDefaultPrm.stMovRelPrm;
stMovRelPrm.fDistance := fDistance;
stMovRelPrm.fVelocity := fVelocity;
stMovRelPrm.fAcceleration := fAcceleration;
stMovRelPrm.fDeceleration := fDeceleration;

eCommandRequest := E_MotionCommand.eMotionCommand_moveRel;
MoveRelAccDec := E_OperationResult.eOperationResult_Ok;
END_METHOD

/// Performs an relative axis positioning using specified parameter set.
/// This motion is capable to overlay (max. 2 parallel at one time)
{attribute 'object_name' := 'MoveRelEx'}
METHOD MoveRelEx : E_OperationResult
VAR_INPUT
	/// Parameter set to use
	stMovRelParameter: ST_AxisMoveRelParameter;
END_VAR
// move axis rel

MoveRelEx := THIS^.MoveRel(stMovRelParameter.fDistance);

IF MoveRelEx = E_OperationResult.eOperationResult_Ok THEN
	stMovRelPrm := stMovRelParameter;
END_IF
END_METHOD

/// Performs an relative axis positioning using specified parameter set.
/// This motion is capable to overlay (max. 2 parallel at one time)
{attribute 'object_name' := 'MoveRelExVel'}
METHOD MoveRelExVel : E_OperationResult
VAR_INPUT
	/// Distance to move to
	fDistance: LREAL;
	/// Speed
	fVelocity: LREAL;
END_VAR
// move axis rel

// init result pessimistic
MoveRelExVel := E_OperationResult.eOperationResult_NOk;

// if stopping or resetting is active return --> higher prio
IF eCommandExecute = E_MotionCommand.eMotionCommand_reset OR eCommandExecute = E_MotionCommand.eMotionCommand_stop THEN
	RETURN;
END_IF

stMovRelPrm := stDefaultPrm.stMovRelPrm;
stMovRelPrm.fDistance := fDistance;
stMovRelPrm.fVelocity := fVelocity;

eCommandRequest := E_MotionCommand.eMotionCommand_moveRel;
MoveRelExVel := E_OperationResult.eOperationResult_Ok;
END_METHOD

/// Performs an velocity axis movement using default parameter set.
/// This motion is capable to overlay (max. 2 parallel at one time)
{attribute 'object_name' := 'MoveVel'}
METHOD MoveVel : E_OperationResult
VAR_INPUT
	/// Velocity
	fVelocity: LREAL;
	/// Direction
	eDirection: TC2_MC2.MC_Direction;
END_VAR
// move axis vel

// init result pessimistic
MoveVel := E_OperationResult.eOperationResult_NOk;

// if stopping or resetting is active return --> higher prio
IF eCommandExecute = E_MotionCommand.eMotionCommand_reset OR eCommandExecute = E_MotionCommand.eMotionCommand_stop THEN
	RETURN;
END_IF

stMovVelPrm := stDefaultPrm.stMovVelPrm;
stMovVelPrm.fVelocity := fVelocity;
stMovVelPrm.eDirection := eDirection;

eCommandRequest := E_MotionCommand.eMotionCommand_moveVel;
MoveVel := E_OperationResult.eOperationResult_Ok;
END_METHOD

/// Performs an velocity axis movement using default parameter set.
/// This motion is capable to overlay (max. 2 parallel at one time)
{attribute 'object_name' := 'MoveVelAccDec'}
METHOD MoveVelAccDec : E_OperationResult
VAR_INPUT
	/// Velocity
	fVelocity: LREAL;
	/// Direction
	eDirection: TC2_MC2.MC_Direction;
	/// Acceleration
	fAcceleration	: LREAL;
	/// Deceleration
	fDeceleration	: LREAL;	
END_VAR
// move axis vel

// init result pessimistic
MoveVelAccDec := E_OperationResult.eOperationResult_NOk;

// if stopping or resetting is active return --> higher prio
IF eCommandExecute = E_MotionCommand.eMotionCommand_reset OR eCommandExecute = E_MotionCommand.eMotionCommand_stop THEN
	RETURN;
END_IF

stMovVelPrm := stDefaultPrm.stMovVelPrm;
stMovVelPrm.fVelocity := fVelocity;
stMovVelPrm.eDirection := eDirection;
stMovVelPrm.fAcceleration := fAcceleration;
stMovVelPrm.fDeceleration := fDeceleration;

eCommandRequest := E_MotionCommand.eMotionCommand_moveVel;
MoveVelAccDec := E_OperationResult.eOperationResult_Ok;
END_METHOD

/// Performs an velocity axis movement using specified parameter
/// This motion is capable to overlay (max. 2 parallel at one time)
{attribute 'object_name' := 'MoveVelEx'}
METHOD MoveVelEx : E_OperationResult
VAR_INPUT
	/// Parameter set to use
	stMovVelParameter: ST_AxisMoveVelParameter;
END_VAR
// move axis abs

MoveVelEx := THIS^.MoveVel(stMovVelParameter.fVelocity, stMovVelParameter.eDirection);

IF MoveVelEx = E_OperationResult.eOperationResult_Ok THEN
	stMovVelPrm := stMovVelParameter;
END_IF
END_METHOD

{attribute 'monitoring' := 'call'}
PROPERTY Moving : BOOL
GET
Moving := fbAxisRef.Status.Moving;
END_GET
END_PROPERTY

{attribute 'monitoring' := 'call'}
PROPERTY NotMoving : BOOL
GET
NotMoving := fbAxisRef.Status.NotMoving;
END_GET
END_PROPERTY

{attribute 'monitoring' := 'call'}
PROPERTY Override : LREAL
GET
Override := fSetOverride;
END_GET
SET
fSetOverride := LIMIT(0, Override, 100);
END_SET
END_PROPERTY

/// Get's a value, indicating whether axis position is in target position or higher.
METHOD PUBLIC PositionReachedOrHigher : BOOL
VAR_INPUT
	fPosition	: LREAL;
END_VAR
PositionReachedOrHigher := Position >= (fPosition - fEpsilon);
END_METHOD

/// Get's a value, indicating whether axis position is in target position or lower.
METHOD PUBLIC PositionReachedOrLower : BOOL
VAR_INPUT
	fPosition	: LREAL;
END_VAR
PositionReachedOrLower := Position <= (fPosition + fEpsilon);
END_METHOD

/// Get's a value, indicating whether axis position is in target position window.
METHOD PUBLIC PositionReachedWindow : BOOL
VAR_INPUT
	fPosition	: LREAL;
	fWindow 	: LREAL;
END_VAR
PositionReachedWindow := ABS(Position - fPosition) <= fWindow AND NotMoving;
END_METHOD

/// Reset component logic
{attribute '' := ''}
{attribute 'object_name' := 'Reset'}
METHOD Reset
// base logic run
SUPER^.Reset();

// reset axis
tonTimeout(IN := FALSE);
eCommandRequest := E_MotionCommand.eMotionCommand_reset;
eState := E_ComponentState.eComponentState_resetting;

nErrorId := 0;
END_METHOD

/// Forces MC reset (e.g.: reset lag distance)
METHOD ResetMc : E_OperationResult
// set axis pos

// init result pessimistic
ResetMc := E_OperationResult.eOperationResult_NOk;

// if stopping or resetting is active return --> higher prio
IF eCommandExecute = E_MotionCommand.eMotionCommand_reset OR eCommandExecute = E_MotionCommand.eMotionCommand_stop THEN
	RETURN;
END_IF

eCommandRequest := eMotionCommand_resetMc;

ResetMc := E_OperationResult.eOperationResult_Ok;
END_METHOD

/// Run component logic
{attribute 'object_name' := 'Run'}
METHOD Run : E_ComponentState
// base logic run
Run := SUPER^.Run();

// return here as long axis ref not set
IF NOT __ISVALIDREF(fbAxisRef) THEN
	//aSClearText[0] := 'Axis ref not set!';
	//aSClearText := F_GetTranslatedTxtLib("Axis ref not set!", eLanguage);
	RETURN;
END_IF

// switch case request
CASE eCommandRequest OF	
	/// No command
	E_MotionCommand.eMotionCommand_none:
	
	/// Reset axis
	E_MotionCommand.eMotionCommand_reset, eMotionCommand_resetMc:
		IF (eCommandExecute <> E_MotionCommand.eMotionCommand_stop AND eCommandExecute <> E_MotionCommand.eMotionCommand_halt) OR fbAxisRef.Status.StandStill THEN
			eCommandExecute := eCommandRequest;
			eCommandRequest := E_MotionCommand.eMotionCommand_none;
		END_IF
	
	/// Axis halt (default stopping method)
	E_MotionCommand.eMotionCommand_halt:
		IF eCommandExecute <> E_MotionCommand.eMotionCommand_stop THEN
			eCommandExecute := eCommandRequest;
			eCommandRequest := E_MotionCommand.eMotionCommand_none;
		END_IF;
	
	/// Axis stop (needs reset before next motion command)
	E_MotionCommand.eMotionCommand_stop:
		eCommandExecute := eCommandRequest;
		eCommandRequest := E_MotionCommand.eMotionCommand_none;
	
	/// other commands
	E_MotionCommand.eMotionCommand_home,
	E_MotionCommand.eMotionCommand_jog,
	E_MotionCommand.eMotionCommand_jogAcc,
	E_MotionCommand.eMotionCommand_moveAbs,
	E_MotionCommand.eMotionCommand_moveAdd,
	E_MotionCommand.eMotionCommand_moveRel,
	E_MotionCommand.eMotionCommand_moveMod,
	E_MotionCommand.eMotionCommand_moveVel,
	E_MotionCommand.eMotionCommand_torque,
	E_MotionCommand.eMotionCommand_gearIn,
	E_MotionCommand.eMotionCommand_gearOut,
	E_MotionCommand.eMotionCommand_touchProbe,
	E_MotionCommand.eMotionCommand_torqCtrl:
		// wait for active command none and axis ready
		IF eCommandExecute = eMotionCommand_none AND fbPower.Status THEN
			eCommandExecute := eCommandRequest;
			eCommandRequest := E_MotionCommand.eMotionCommand_none;
		END_IF
		
	E_MotionCommand.eMotionCommand_setPos,
	E_MotionCommand.eMotionCommand_setAxPosOffs:
		IF eCommandExecute = eMotionCommand_none THEN
			eCommandExecute := eCommandRequest;
			eCommandRequest := E_MotionCommand.eMotionCommand_none;
		END_IF
	
END_CASE

// call workflows 
WfDiagnostic();
WfPower();
WfReset();
WfHome();
WfSetPos();
WfJog();
WfJogAcc();
WfMovAbs();
WfMovAdd();
WfMovRel();
WfMovMod();
WfMovVel();
WfGearIn();
WfGearOut();
WfTorqCtrl();
WfHalt();
WfStop();
WfErrorHandling();
WfSoE();
WfInitPositionOffset();
WfAxSetPosOffset();

// set clear text
IF eState <> E_ComponentState.eComponentState_error THEN
	;
ELSE
	aSClearText := F_CreateDynText( WConcat("error number: ", UDINT_TO_WSTRING(nErrorID)), 0);
	// try get details
	IF eAxisType = E_AxisType.AX5xxx THEN
		IF fbAxisRef.Status.Error AND stAX5xxxDiag.stDiagNumberList.arrDiagNumbers[0] <> 0 THEN
			sMsg := stAX5xxxDiag.strDiagMessage; // display diag msg
			FOR ii := 0 TO 2 DO	// add first 3 error codes 
				sMsg := Concat3(sMsg, ', ', UDINT_TO_STRING(stAX5xxxDiag.stDiagNumberList.arrDiagNumbers[ii]));
			END_FOR
			aSClearText.wsName := STRING_TO_WSTRING(sMsg);
		END_IF
	// Bosch Indradrive
	ELSIF eAxisType = E_AxisType.Bosch_IndradriveEc THEN
		sMsg := stIndraDrvDiag.strDiagMessage; // display diag msg
		FOR ii := 0 TO 2 DO	// add first 3 error codes 
			sMsg := Concat3(sMsg, ', ', UDINT_TO_STRING(stIndraDrvDiag.stDiagNumberList.arrDiagNumbers[ii]));
		END_FOR
		aSClearText.wsName := STRING_TO_WSTRING(sMsg);
		
	END_IF
END_IF

// Ausgabedaten
bError := (eState = E_ComponentState.eComponentState_error);
Position := fbAxisRef.NcToPlc.ActPos;
ModuloPosition := fbAxisRef.NcToPlc.ModuloActPos;
Operational := fbAxisRef.Status.Operational AND NOT fbAxisRef.Status.Disabled;
fPosDiff := fbAxisRef.NcToPlc.PosDiff;
Homed := fbAxisRef.Status.Homed;
bHasJob := fbAxisRef.Status.HasJob;
bHoldActiv := bHold;
bHold := FALSE;

CheckLatchState();
END_METHOD

/// Set axis reference
{attribute 'object_name' := 'SetAxisReference'}
METHOD SetAxisReference
VAR_IN_OUT
	/// NC Axis reference
	fbRefAxis: AXIS_REF;
	/// Additional inputs from axis
	stRefIn: ST_AxisIn;
	/// Additional outputs to axis
	stRefOut: ST_AxisOut;
END_VAR
fbAxisRef REF= fbRefAxis;
stIn REF= stRefIn;
stOut REF= stRefOut;
END_METHOD

/// Set axis position, method with minimal options
{attribute 'object_name' := 'SetAxPosOffs'}
METHOD SetAxPosOffs : E_OperationResult
VAR_INPUT
	/// Parameter set to use
	fPosition 	: REAL;
END_VAR
// set ax axis pos offset

// init result pessimistic
SetAxPosOffs := SetAxPosOffsEx(fPosition, FALSE, 
					E_PositionOffsetFeedback.ePositionOffsetFeedback1, 
					E_PositionOffsetMemory.ePositionOffsetMemory_Drive);
END_METHOD

/// Set axis position, extended method with all options
{attribute 'object_name' := 'SetAxPosOffsEx'}
METHOD SetAxPosOffsEx : E_OperationResult
VAR_INPUT
	/// Parameter set to use
	fPosition 	: REAL;
	bRelative 	: BOOL;
	eFeedback 	: E_PositionOffsetFeedback;
	eMemory 	: E_PositionOffsetMemory;
END_VAR
// set ax axis pos offset

// init result pessimistic
SetAxPosOffsEx := E_OperationResult.eOperationResult_NOk;

// if stopping or resetting is active return --> higher prio
IF eCommandExecute = E_MotionCommand.eMotionCommand_reset OR eCommandExecute = E_MotionCommand.eMotionCommand_stop THEN
	RETURN;
END_IF

fbAxSetPosOffs.Position := fPosition;
fbAxSetPosOffs.Relative := bRelative;
fbAxSetPosOffs.Feedback := eFeedback;
fbAxSetPosOffs.Memory := eMemory;

eCommandRequest := E_MotionCommand.eMotionCommand_setAxPosOffs;
SetAxPosOffsEx := E_OperationResult.eOperationResult_Ok;
END_METHOD

/// Axis home reset
{attribute 'object_name' := 'SetCalibration'}
METHOD SetCalibration : E_OperationResult
VAR_INPUT
	/// TRUE = Set-Calibration, FALSE = Reset-Calibration
	bSet			:BOOL;
END_VAR
// home axis

SetCalibration := THIS^.Home();

IF SetCalibration = E_OperationResult.eOperationResult_Ok THEN
	IF bSet THEN
		stHomingPrm.eHomingMode := MC_HomingMode.MC_ForceCalibration;		
	ELSE
		stHomingPrm.eHomingMode := MC_HomingMode.MC_ResetCalibration;
	END_IF
END_IF
END_METHOD

/// Set axis position
{attribute 'object_name' := 'SetPos'}
METHOD SetPos : E_OperationResult
VAR_INPUT
	fPosition: LREAL;
END_VAR
// set axis pos

// init result pessimistic
SetPos := E_OperationResult.eOperationResult_NOk;

// if stopping or resetting is active return --> higher prio
IF eCommandExecute = E_MotionCommand.eMotionCommand_reset OR eCommandExecute = E_MotionCommand.eMotionCommand_stop THEN
	RETURN;
END_IF

stSetPosPrm := stDefaultPrm.stSetPosPrm;
stSetPosPrm.fPosition := fPosition;

eCommandRequest := E_MotionCommand.eMotionCommand_setPos;
SetPos := E_OperationResult.eOperationResult_Ok;
END_METHOD

/// Set axis position, extended method with all options
{attribute 'object_name' := 'SetPosEx'}
METHOD SetPosEx : E_OperationResult
VAR_INPUT
	/// Parameter set to use
	stSetPosParameter: ST_AxisSetPosParameter;
END_VAR
// set axis pos

SetPosEx := THIS^.SetPos(stSetPosParameter.fPosition);

IF SetPosEx = E_OperationResult.eOperationResult_Ok THEN
	stSetPosPrm := stSetPosParameter;
END_IF
END_METHOD

/// Set axis position SoE for Indra drives
METHOD SetPosIndraSoE : E_OperationResult
VAR_INPUT
	fPosition: LREAL;
END_VAR
// set axis pos

// init result pessimistic
SetPosIndraSoE := E_OperationResult.eOperationResult_NOk;

// if stopping or resetting is active return --> higher prio
IF eCommandExecute = E_MotionCommand.eMotionCommand_reset OR eCommandExecute = E_MotionCommand.eMotionCommand_stop THEN
	RETURN;
END_IF

stSoE.fRealValue := LREAL_TO_REAL(fPosition * 1E-4);
stSoE.eCmd := E_SoECommand.eSoECommand_writeIndraDrvPos;

SetPosIndraSoE := E_OperationResult.eOperationResult_Ok;
END_METHOD

/// Axis stop using default parameter
{attribute 'object_name' := 'Stop'}
METHOD Stop : E_OperationResult
// stop axis

stStopPrm := stDefaultPrm.stStopPrm;

eCommandRequest := E_MotionCommand.eMotionCommand_stop;
Stop := E_OperationResult.eOperationResult_Ok;
// sofort aufrufen
Run();
END_METHOD

/// Axis stop using specified parameter
{attribute 'object_name' := 'StopEx'}
METHOD StopEx : E_OperationResult
VAR_INPUT
	/// Parameter set to use
	stStopParameter: ST_AxisStopParameter;
END_VAR
// stop axis

stStopPrm := stStopParameter;
StopEx := THIS^.Stop();
END_METHOD

/// Get's a value, indicating whether axis position is within target position window and not moving.
/// Position window: default epsilon (1E-3).
/// Valid for previous ABS movement's.
METHOD PUBLIC TargetReached : BOOL
VAR_INPUT
END_VAR
TargetReached := TargetWindowReached(fEpsilon);
END_METHOD

/// Get's a value, indicating whether axis position is within target position window and not moving.
/// Extended: timeout
/// Position window: default epsilon (1E-3).
/// Valid for previous ABS movement's.
METHOD PUBLIC TargetReachedEx : BOOL
VAR_INPUT
	tTimeout	: TIME;
END_VAR
TargetReachedEx := TargetWindowReachedEx(fEpsilon, tTimeout);
END_METHOD

/// Get's a value, indicating whether axis position is within target position window and not moving.
/// Valid for previous ABS movement's. 
METHOD PUBLIC TargetWindowReached : BOOL
VAR_INPUT
	fWindow : LREAL;
END_VAR
TargetWindowReached := Position >= (stMovAbsPrm.fPosition - fWindow) AND Position <= (stMovAbsPrm.fPosition + fWindow) AND NotMoving;
END_METHOD

/// Get's a value, indicating whether axis position is within target position window and not moving.
/// Extended: timeout
/// Valid for previous ABS movement's. 
METHOD PUBLIC TargetWindowReachedEx : BOOL
VAR_INPUT
	fWindow 	: LREAL;
	tTimeout	: TIME;
END_VAR
VAR
	bPosOk		: BOOL;
END_VAR
bPosOk := TargetWindowReached(fWindow);

tonTimeout(IN := NOT bPosOk, PT := tTimeout);
IF tonTimeout.Q THEN
	M_SetLocalError(F_CreateDynText("Zeitueberschreitung bei Positionierung", 0));
	Halt();
	bError := TRUE;
END_IF

TargetWindowReachedEx := bPosOk;
END_METHOD

{attribute 'object_name' := 'TorqCtrl'}
METHOD TorqCtrl : E_OperationResult
VAR_INPUT
	/// torque value [%]
	fTorque: LREAL;
END_VAR
// axis in torque control mode

// init result pessimistic
TorqCtrl := E_OperationResult.eOperationResult_NOk;

// if stopping or resetting is active return --> higher prio
IF eCommandExecute = E_MotionCommand.eMotionCommand_reset OR eCommandExecute = E_MotionCommand.eMotionCommand_stop THEN
	RETURN;
END_IF

stTorqCtrlPrm := stDefaultPrm.stTorqCtrlPrm;
stTorqCtrlPrm.fTorque := fTorque;

eCommandRequest := E_MotionCommand.eMotionCommand_torqCtrl;
TorqCtrl := E_OperationResult.eOperationResult_Ok;
END_METHOD

{attribute 'object_name' := 'TorqCtrlEx'}
METHOD TorqCtrlEx : E_OperationResult
VAR_INPUT
	/// Parameter set to use
	stParameter: ST_AxisTorqCtrlParameter;
END_VAR
// axis in torque control mode

TorqCtrlEx := THIS^.TorqCtrl(stParameter.fTorque);

IF TorqCtrlEx = E_OperationResult.eOperationResult_Ok THEN
	stTorqCtrlPrm := stParameter;
END_IF
END_METHOD

/// Actual torque [Nm]
{attribute 'monitoring' := 'call'}
PROPERTY Torque : LREAL
GET
/// Actual torque [Nm]
Torque := fbAxisRef.NcToPlc.ActTorque * fTorqueFactor;
END_GET
END_PROPERTY

/// The torque limit for both directions. [%]
{attribute 'monitoring' := 'call'}
PROPERTY TorqueLimit : LREAL
GET
/// The torque limit for both directions. [0.1%]
TorqueLimit := INT_TO_LREAL(stOut.iBipolarTorqueLimitValue);
END_GET
SET
stOut.iBipolarTorqueLimitValue := LREAL_TO_INT(TorqueLimit);
END_SET
END_PROPERTY

{attribute 'monitoring' := 'call'}
PROPERTY Velocity : LREAL
GET
Velocity  := fbAxisRef.NcToPlc.ActVelo;
END_GET
END_PROPERTY

ACTION WfAxSetPosOffset:

/// Workflow set ax position offset

// call fb cyclic
//fbAxSetPosOffs.Position := fPosition;
//fbAxSetPosOffs.Relative := bRelative;
//fbAxSetPosOffs.Feedback := E_PositionOffsetFeedback.ePositionOffsetFeedback1;
//fbAxSetPosOffs.Memory := E_PositionOffsetMemory.ePositionOffsetMemory_Drive;
fbAxSetPosOffs(Axis := fbAxisRef);

// FB diagnostic and reset 
IF fbAxSetPosOffs.Execute AND NOT fbAxSetPosOffs.Busy THEN
	IF fbAxSetPosOffs.Error THEN			
		nErrorId := fbAxSetPosOffs.ErrorID;
		M_SetLocalErrorS('Error set ax position offset: ErrId: ', TO_STRING(nErrorId));
	END_IF
	fbAxSetPosOffs.Execute := FALSE;
END_IF

// return if other command active	
IF eCommandExecute <> E_MotionCommand.eMotionCommand_setAxPosOffs THEN
	RETURN;
END_IF

//aSClearText := F_GetTranslatedTxtLib('Set ax position offset', eLanguage);		
IF NOT fbAxSetPosOffs.Busy THEN
	fbAxSetPosOffs(Axis := fbAxisRef, Execute := TRUE);
	eCommandExecute := E_MotionCommand.eMotionCommand_none;
END_IF
END_ACTION

ACTION WfDiagnostic:

/// Workflow axis diagnostic

// run axis FBs
fbAxisRef.ReadStatus();

// return in case of reset
(*IF eCommandExecute = E_MotionCommand.eMotionCommand_reset THEN
	RETURN;
END_IF*)

// diagnostics AX5xxx
IF eAxisType = E_AxisType.AX5xxx THEN
	// Diag + Reset of AX5000
	// call drive diag FBs
	fbAX5xxxDiag(
		IPCNetID	:= IPCNetID,
		Axis		:= fbAxisRef,
		stAX5000Diag:= stAX5xxxDiag);

	// clear reset/diag request if not active
	fbAX5xxxDiag.Reset := fbAX5xxxDiag.Reset AND fbAX5xxxDiag.ResetAct;
	fbAX5xxxDiag.GetDiag := fbAX5xxxDiag.GetDiag AND fbAX5xxxDiag.DiagAct;

	//IF fbAX5xxxDiag.Error THEN... / nErrorId := fbAX5xxxDiag.AdsErrId; -> WfErrorHandling
	stDriveRef := fbAX5xxxDiag.DriveRef;
	
// Bosch Indradrive
ELSIF eAxisType = E_AxisType.Bosch_IndradriveEc THEN
	// Diag + Reset of Indradrive
	// call drive diag FBs
	fbIndraDrvDiag(
		sIPCNetID	:= IPCNetID,
		Axis		:= fbAxisRef,
		stDriveDiag:= stIndraDrvDiag);

	// clear reset/diag request if not active
	fbIndraDrvDiag.bReset := fbIndraDrvDiag.bReset AND fbIndraDrvDiag.bResetAct;
	fbIndraDrvDiag.bGetDiag := fbIndraDrvDiag.bGetDiag AND fbIndraDrvDiag.bDiagAct;

	//IF fbAX5xxxDiag.Error THEN... / nErrorId := fbAX5xxxDiag.AdsErrId; -> WfErrorHandling
	stDriveRef := fbIndraDrvDiag.stDriveRef;
END_IF
END_ACTION

ACTION WfErrorHandling:

// chk axis operational
tonChkOperation(IN := (eState = E_ComponentState.eComponentState_running AND fbPower.Enable AND 
						NOT fbAxisRef.Status.Operational), PT := T#5S);
IF tonChkOperation.Q THEN
	eState := E_ComponentState.eComponentState_error;
END_IF
// Safety Error liegt an
IF bAX5805_Error AND eAxisType = E_AxisType.AX5xxx THEN
	M_SetLocalError(CONST.stTextListGlobal.stText_Comp.stText_Axis_SafetyError);
END_IF

// run error trigger
rtrigError(CLK := fbAxisRef.Status.Error OR stAX5xxxDiag.bAxisError OR stIndraDrvDiag.bAxisError OR
					eState = E_ComponentState.eComponentState_error);
IF rtrigError.Q THEN
	eState := E_ComponentState.eComponentState_error;
	// AX5000
	IF eAxisType = E_AxisType.AX5xxx THEN
		IF fbAxisRef.Status.Error AND fbAxisRef.Status.ErrorID = 18000 THEN
			bErrDiagActive := TRUE;
			fbAX5xxxDiag.GetDiag := TRUE; // get diag for AX5xxx
		ELSE
			IF tonChkOperation.Q THEN	
				M_SetLocalError(CONST.stTextListGlobal.stText_Comp.stText_Axis_DriveNotReady);
			ELSIF bAX5805_Error THEN
				M_SetLocalError(CONST.stTextListGlobal.stText_Comp.stText_Axis_SafetyError);
			ELSIF nErrorId = 16931 THEN
				M_SetLocalError(CONST.stTextListGlobal.stText_Comp.stText_Axis_MovingNotReleased);
			ELSIF nErrorId = 17505 THEN
				M_SetLocalError(CONST.stTextListGlobal.stText_Comp.stText_Axis_TargetOutOfArea);
			ELSIF nErrorId = 18000 THEN
				M_SetLocalError(CONST.stTextListGlobal.stText_Comp.stText_Axis_HwNotReady);
			ELSIF nErrorId <> 0 THEN
				M_SetLocalErrorEx(CONST.stTextListGlobal.stText_Comp.stText_Axis_FbError, F_CreateDynText(TO_WSTRING(nErrorId), 0));
			ELSIF fbAxisRef.Status.ErrorID <> 0 THEN
				M_SetLocalErrorEx(CONST.stTextListGlobal.stText_Comp.stText_Axis_NcError, F_CreateDynText(TO_WSTRING(fbAxisRef.Status.ErrorID), 0));
			END_IF	
		END_IF	
	
	// Bosch Indradrive
	ELSIF eAxisType = E_AxisType.Bosch_IndradriveEc THEN
		IF fbAxisRef.Status.Error AND fbAxisRef.Status.ErrorID = 18000 THEN
			bErrDiagActive := TRUE;
			fbIndraDrvDiag.bGetDiag := TRUE; // get diag for Indradrive
		ELSE
			IF tonChkOperation.Q THEN	
				M_SetLocalError(CONST.stTextListGlobal.stText_Comp.stText_Axis_DriveNotReady);
			ELSIF bAX5805_Error THEN
				M_SetLocalError(CONST.stTextListGlobal.stText_Comp.stText_Axis_SafetyError);
			ELSIF nErrorId = 16931 THEN
				M_SetLocalError(CONST.stTextListGlobal.stText_Comp.stText_Axis_MovingNotReleased);
			ELSIF nErrorId = 17505 THEN
				M_SetLocalError(CONST.stTextListGlobal.stText_Comp.stText_Axis_TargetOutOfArea);
			ELSIF nErrorId = 18000 THEN
				M_SetLocalError(CONST.stTextListGlobal.stText_Comp.stText_Axis_HwNotReady);
			ELSIF nErrorId <> 0 THEN
				M_SetLocalErrorEx(CONST.stTextListGlobal.stText_Comp.stText_Axis_FbError, F_CreateDynText(TO_WSTRING(nErrorId), 0));
			ELSIF fbAxisRef.Status.ErrorID <> 0 THEN
				M_SetLocalErrorEx(CONST.stTextListGlobal.stText_Comp.stText_Axis_NcError, F_CreateDynText(TO_WSTRING(fbAxisRef.Status.ErrorID), 0));
			END_IF
		END_IF

	ELSE
		IF nErrorId <> 0 THEN
			M_SetLocalErrorEx(CONST.stTextListGlobal.stText_Comp.stText_Axis_FbError, F_CreateDynText(TO_WSTRING(nErrorId), 0));
		ELSIF fbAxisRef.Status.ErrorID <> 0 THEN
			M_SetLocalErrorEx(CONST.stTextListGlobal.stText_Comp.stText_Axis_NcError, F_CreateDynText(TO_WSTRING(fbAxisRef.Status.ErrorID), 0));
		END_IF
	END_IF
END_IF


// run AX5000 diag 
ftrigDiag(CLK := fbAX5xxxDiag.DiagAct);
IF ftrigDiag.Q AND bErrDiagActive THEN
	bErrDiagActive := FALSE;
	IF fbAxisRef.Status.Error AND stAX5xxxDiag.stDiagNumberList.arrDiagNumbers[0] <> 0 THEN
		sMsg := Concat3(TO_STRING(stName.wsName), ': ', stAX5xxxDiag.strDiagMessage); // display diag msg
		FOR ii := 0 TO 2 DO	// add first 3 error codes 
			sMsg := Concat3(sMsg, ', ', UDINT_TO_STRING(stAX5xxxDiag.stDiagNumberList.arrDiagNumbers[ii]));
		END_FOR
		M_SetLocalErrorEx(CONST.stTextListGlobal.stText_Comp.stText_Axis_HwError, F_CreateDynText(TO_WSTRING(sMsg), 0));

	ELSE
		sMsg := Concat3(TO_STRING(stName.wsName), ': ', sLastError);
		sMsg := Concat3(sMsg, ' / FehlerNr: ', UDINT_TO_STRING(nErrorId));
		M_SetLocalErrorEx(CONST.stTextListGlobal.stText_Comp.stText_Axis_HwError, F_CreateDynText(TO_WSTRING(sMsg), 0));
	END_IF
END_IF;

// Bosch Indradrive diag
ftrigDiagIndradrv(CLK := fbIndraDrvDiag.bDiagAct);
IF ftrigDiagIndradrv.Q AND bErrDiagActive THEN
	bErrDiagActive := FALSE;
	IF fbAxisRef.Status.Error THEN
		sMsg := Concat3(TO_STRING(stName.wsName), ': ', stIndraDrvDiag.strDiagMessage); // display diag msg
		FOR ii := 0 TO 2 DO	// add first 3 error codes 
			sMsg := Concat3(sMsg, ', ', UDINT_TO_STRING(stIndraDrvDiag.stDiagNumberList.arrDiagNumbers[ii]));
		END_FOR
		M_SetLocalErrorEx(CONST.stTextListGlobal.stText_Comp.stText_Axis_HwError, F_CreateDynText(TO_WSTRING(sMsg), 0));

	ELSE
		sMsg := Concat3(TO_STRING(stName.wsName), ': ', sLastError);
		sMsg := Concat3(sMsg, ' / FehlerNr: ', UDINT_TO_STRING(nErrorId));
		M_SetLocalErrorEx(CONST.stTextListGlobal.stText_Comp.stText_Axis_HwError, F_CreateDynText(TO_WSTRING(sMsg), 0));
	END_IF	
END_IF
END_ACTION

ACTION WfGearIn:

/// Workflow gear in

// call fb cyclic
fbGearIn.GearRatio := stGearInPrm.fGearRatio;
fbGearIn.Acceleration := stGearInPrm.fAcceleration;
fbGearIn.Deceleration := stGearInPrm.fDeceleration;
fbGearIn.Jerk := stGearInPrm.fJerk;
fbGearIn.BufferMode := stGearInPrm.eBufferMode;
fbGearIn.Options := stGearInPrm.stOptions;
IF __ISVALIDREF(stGearInPrm.fbMaster) THEN
	fbGearIn(Master := stGearInPrm.fbMaster, Slave := fbAxisRef);	
END_IF

// FB diagnostic and reset 
IF fbGearIn.Enable AND NOT fbGearIn.Busy THEN
	IF fbGearIn.Error THEN			
		nErrorId := fbGearIn.ErrorID;
		M_SetLocalErrorS('error engine couple: ErrId: ', TO_STRING(nErrorId));
	END_IF
	fbGearIn.Enable := FALSE;
END_IF

// set master axis ID
eMasterAxisId := SEL(fbAxisRef.Status.Coupled, eAxis_none, stGearInPrm.eMasterId);

// return if other command active	
IF eCommandExecute <> E_MotionCommand.eMotionCommand_gearIn THEN
	RETURN;
END_IF

//aSClearText[0] := 'Antrieb Koppeln';	
//aSClearText := F_GetTranslatedTxtLib('engine couple', eLanguage);	
IF NOT fbGearIn.InGear THEN
	fbGearIn.Enable := TRUE;
END_IF
eCommandExecute := E_MotionCommand.eMotionCommand_none;
END_ACTION

ACTION WfGearOut:

/// Workflow gear out

// call fb cyclic
fbGearOut.Options := stGearOutPrm.stOptions;
fbGearOut(Slave := fbAxisRef);

// FB diagnostic and reset 
IF fbGearOut.Execute AND NOT fbGearOut.Busy THEN
	IF fbGearOut.Error THEN
		nErrorId := fbGearOut.ErrorID;
		M_SetLocalErrorS('error engine decouple: ErrId: ', TO_STRING(nErrorId));
	END_IF
	fbGearOut.Execute := FALSE;
END_IF
		
// return if not in gear out
IF eCommandExecute <> E_MotionCommand.eMotionCommand_gearOut THEN
	RETURN;
END_IF

//aSClearText[0] := 'Antrieb Entoppeln';
//aSClearText := F_GetTranslatedTxtEx("engine decouple", eLanguage);
IF stGearOutPrm.bHaltAxis THEN
	stHaltPrm.eBufferMode := MC_Aborting;
	stHaltPrm.fDeceleration := stGearInPrm.fDeceleration;
	stHaltPrm.fJerk := stGearInPrm.fJerk;
	//stHaltPrm.stOptions := stGearInPrm.stOptions;
	THIS^.HaltEx(stHaltPrm);
ELSE
	fbGearOut(Slave := fbAxisRef, Execute := TRUE);	
END_IF
eCommandExecute := E_MotionCommand.eMotionCommand_none;
END_ACTION

ACTION WfHalt:

/// Workflow halting

// call fb cyclic
fbHalt.BufferMode := stHaltPrm.eBufferMode;
fbHalt.Deceleration := stHaltPrm.fDeceleration;
fbHalt.Jerk := stHaltPrm.fJerk;
fbHalt.Options := stHaltPrm.stOptions;
fbHalt(Axis := fbAxisRef);

// FB diagnostic and reset 
IF fbHalt.Execute AND NOT fbHalt.Busy THEN
	IF fbHalt.Error THEN
		nErrorId := fbHalt.ErrorID;
		M_SetLocalErrorS('error at engine halt: ErrId: ', TO_STRING(nErrorId));
	END_IF
	fbHalt.Execute := FALSE;
END_IF
		
// return if not in halting
IF eCommandExecute <> E_MotionCommand.eMotionCommand_halt THEN
	RETURN;
END_IF

//aSClearText[0] := 'Antrieb Halt';
//aSClearText := F_GetTranslatedTxtLib('stop engine', eLanguage);
fbHalt(Axis := fbAxisRef, Execute := TRUE);
eCommandExecute := E_MotionCommand.eMotionCommand_none;
IF fbAxisRef.Status.StandStill THEN
	eCommandExecute := E_MotionCommand.eMotionCommand_none;
END_IF
END_ACTION

ACTION WfHome:

/// Workflow homing

